// TIA Portal V20 export
FUNCTION_BLOCK "LER_AlignThetaCalibration"   // FB101, LAD
// stored: Access Published, MemoryReserve 100, SetENOAutomatically false
   VAR_INPUT
      enable : Bool;
      cmdComplete : Bool;
      AxisXHomePos { ExternalAccessible := 'False'; ExternalVisible := 'False'; ExternalWritable := 'False'} : LReal;
      AxisY1HomePos { ExternalAccessible := 'False'; ExternalVisible := 'False'; ExternalWritable := 'False'} : LReal;
      AxisY2HomePos { ExternalAccessible := 'False'; ExternalVisible := 'False'; ExternalWritable := 'False'} : LReal;
   END_VAR
   VAR_OUTPUT
      Visiontrigger : Bool;
      cmdRequest : Bool;
      error : Bool;
      busy : Bool;
      done : Bool;
      status : Word;
      CmdNummber : DInt;
      CmdParameter1 : DInt;
      CmdParameter2 : DInt;
      CmdParameter3 : DInt;
   END_VAR
   VAR_IN_OUT
      moduleInterface : "LER_typeAlignThetaCalibrationInterface";
      AlignTableAxisX : DB_ANY;
      AlignTableAxisY1 : DB_ANY;
      AlignTableAxisY2 : DB_ANY;
   END_VAR
   VAR
      statAxisXMovePosition : Array[0..18] of LReal;
      statAxisY1MovePosition : Array[0..18] of LReal;
      statAxisY2MovePosition : Array[0..18] of LReal;
      instAlignTableAxisXMCMoveAbs : MC_MOVEABSOLUTE;
      instAlignTableAxisY1MCMoveAbs { S7_SetPoint := 'True'} : MC_MOVEABSOLUTE;
      instAlignTableAxisY2MCMoveAbs { S7_SetPoint := 'True'} : MC_MOVEABSOLUTE;
      statPulse { S7_SetPoint := 'True'} : Array[1..50] of Bool;
      statMoveXCmd : Array[1..10] of Bool;
      statMoveY1Cmd : Array[1..10] of Bool;
      statMoveY2Cmd : Array[1..10] of Bool;
      statVisionCmd : Array[1..10] of Bool;
      statRequstCmd : Array[1..20] of Bool;
      statTimer : Array[1..50] of TON_TIME;
      statAllMoveSeq : DInt;
      statManualMove : Bool;
      statCmdNummber : DInt;
      statCmdParameter1 : DInt;
      statCmdParameter2 : DInt;
      statCmdParameter3 : DInt;
      statPreSeq : DInt;
      statSeqTimeTonTimer : TON_TIME;
   END_VAR
   VAR_TEMP
      tempAlignTableAxisX : REF_TO TO_SynchronousAxis;
      tempAlignTableAxisY1 : REF_TO TO_SynchronousAxis;
      tempAlignTableAxisY2 : REF_TO TO_SynchronousAxis;
      tempAlignTableAxisXPosition : DInt;
      tempAlignTableAxisY1Position : DInt;
      tempAlignTableAxisY2Position : DInt;
   END_VAR
   VAR CONSTANT
      VISION_DELAY_TIME : Time := T#500ms;
      REQ_DELAY_TIME : Time := T#100ms;
   END_VAR
   VAR_TEMP   // added for the SCL form of the ladder/FBD networks
      _w1 : Bool;
      _w2 : Bool;
      _w3 : Bool;
      _w4 : Bool;
      _w5 : Bool;
      _w6 : Bool;
      _w7 : Bool;
      _w8 : Bool;
      _w9 : Bool;
   END_VAR
BEGIN

REGION Network 1 (SCL): Axis Config
   #tempAlignTableAxisX ?= #AlignTableAxisX;
   #tempAlignTableAxisY1 ?= #AlignTableAxisY1;
   #tempAlignTableAxisY2 ?= #AlignTableAxisY2;
END_REGION

REGION Network 2: Teaching Position Config
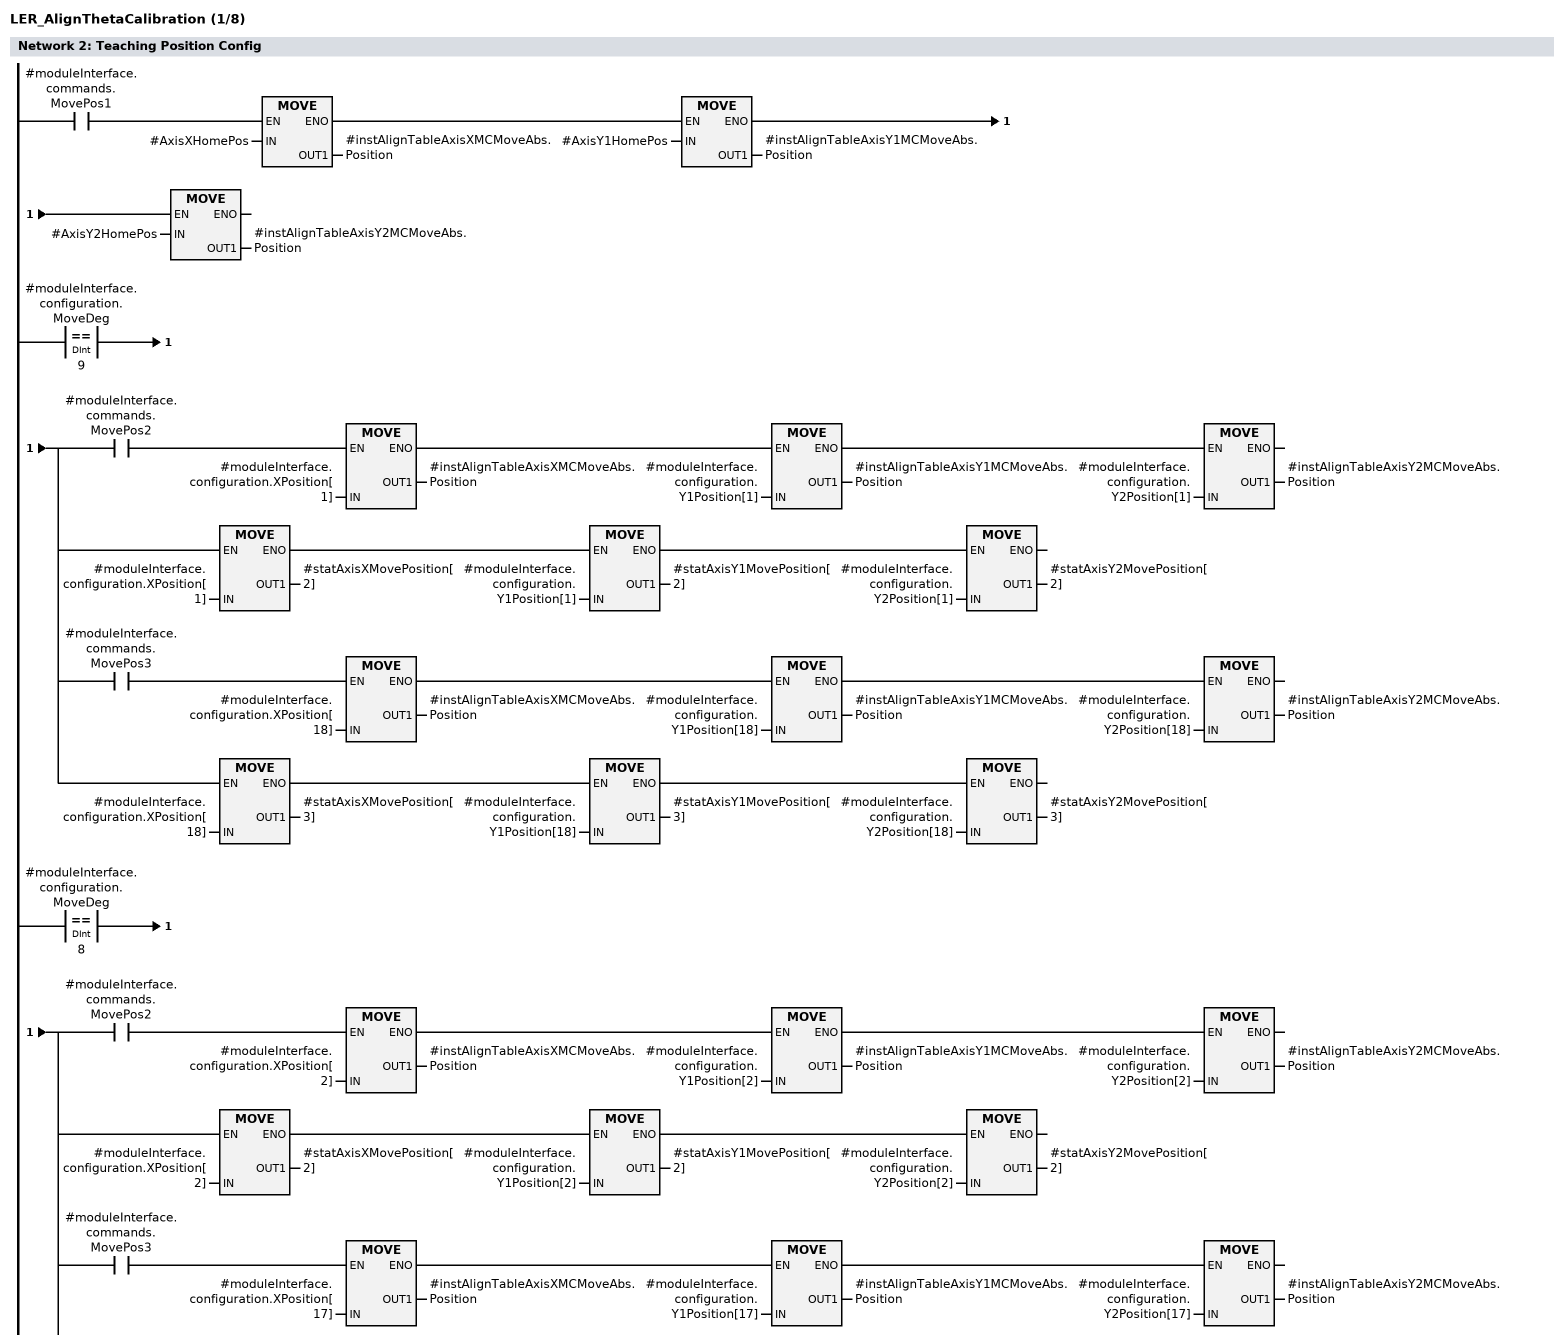
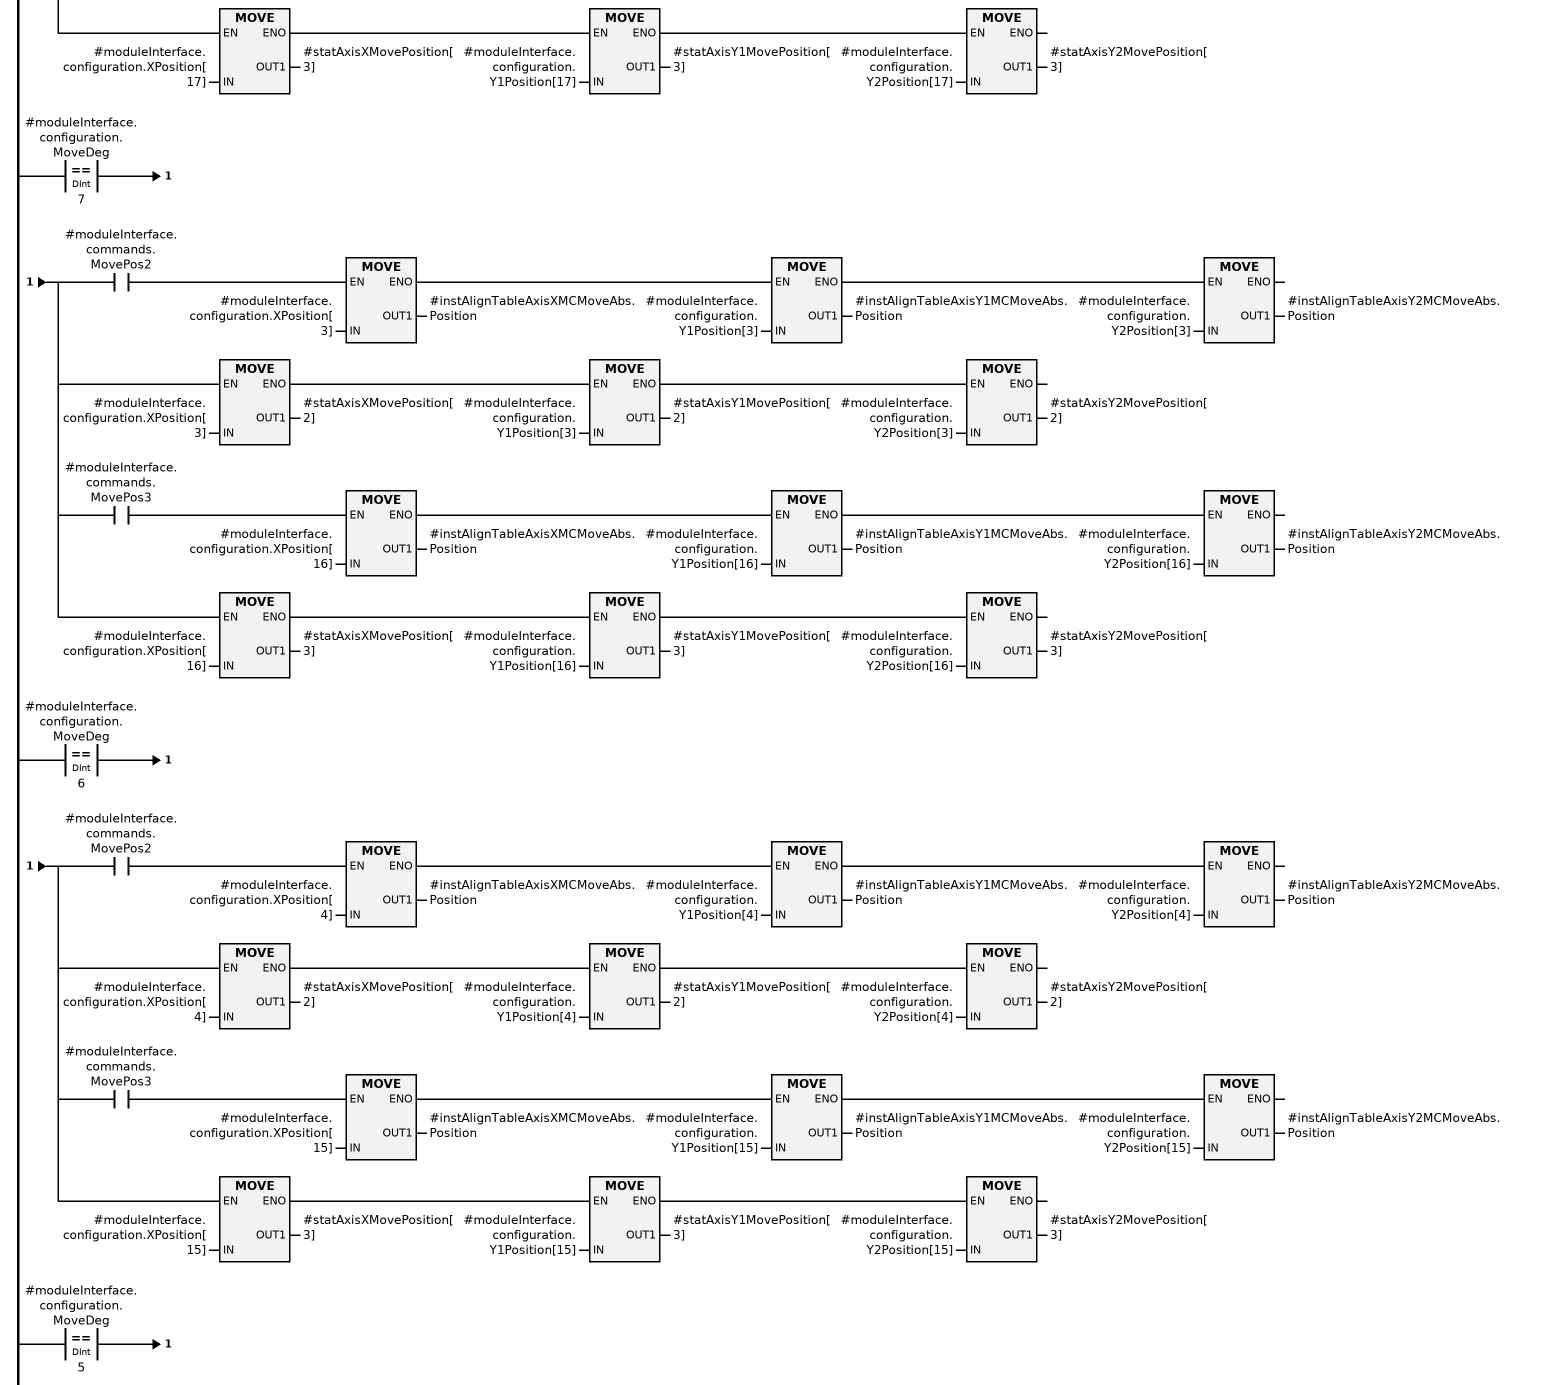
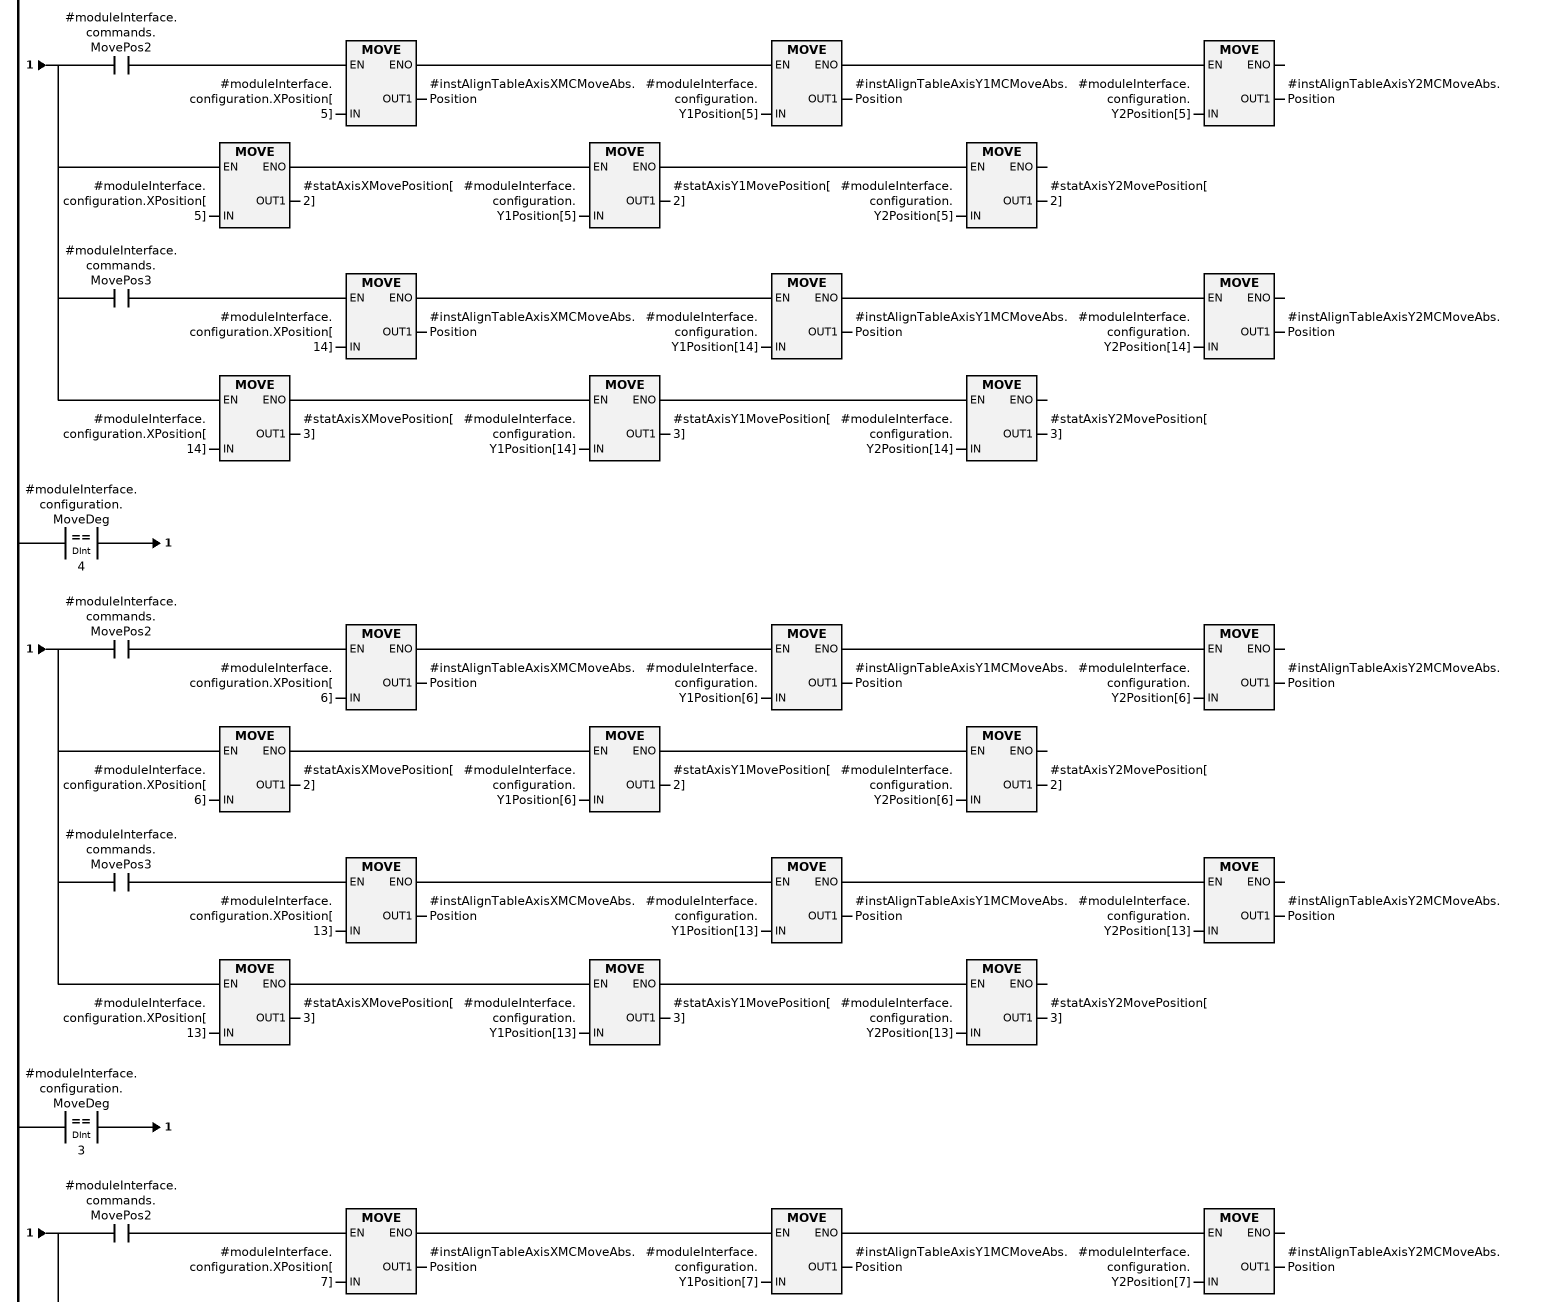
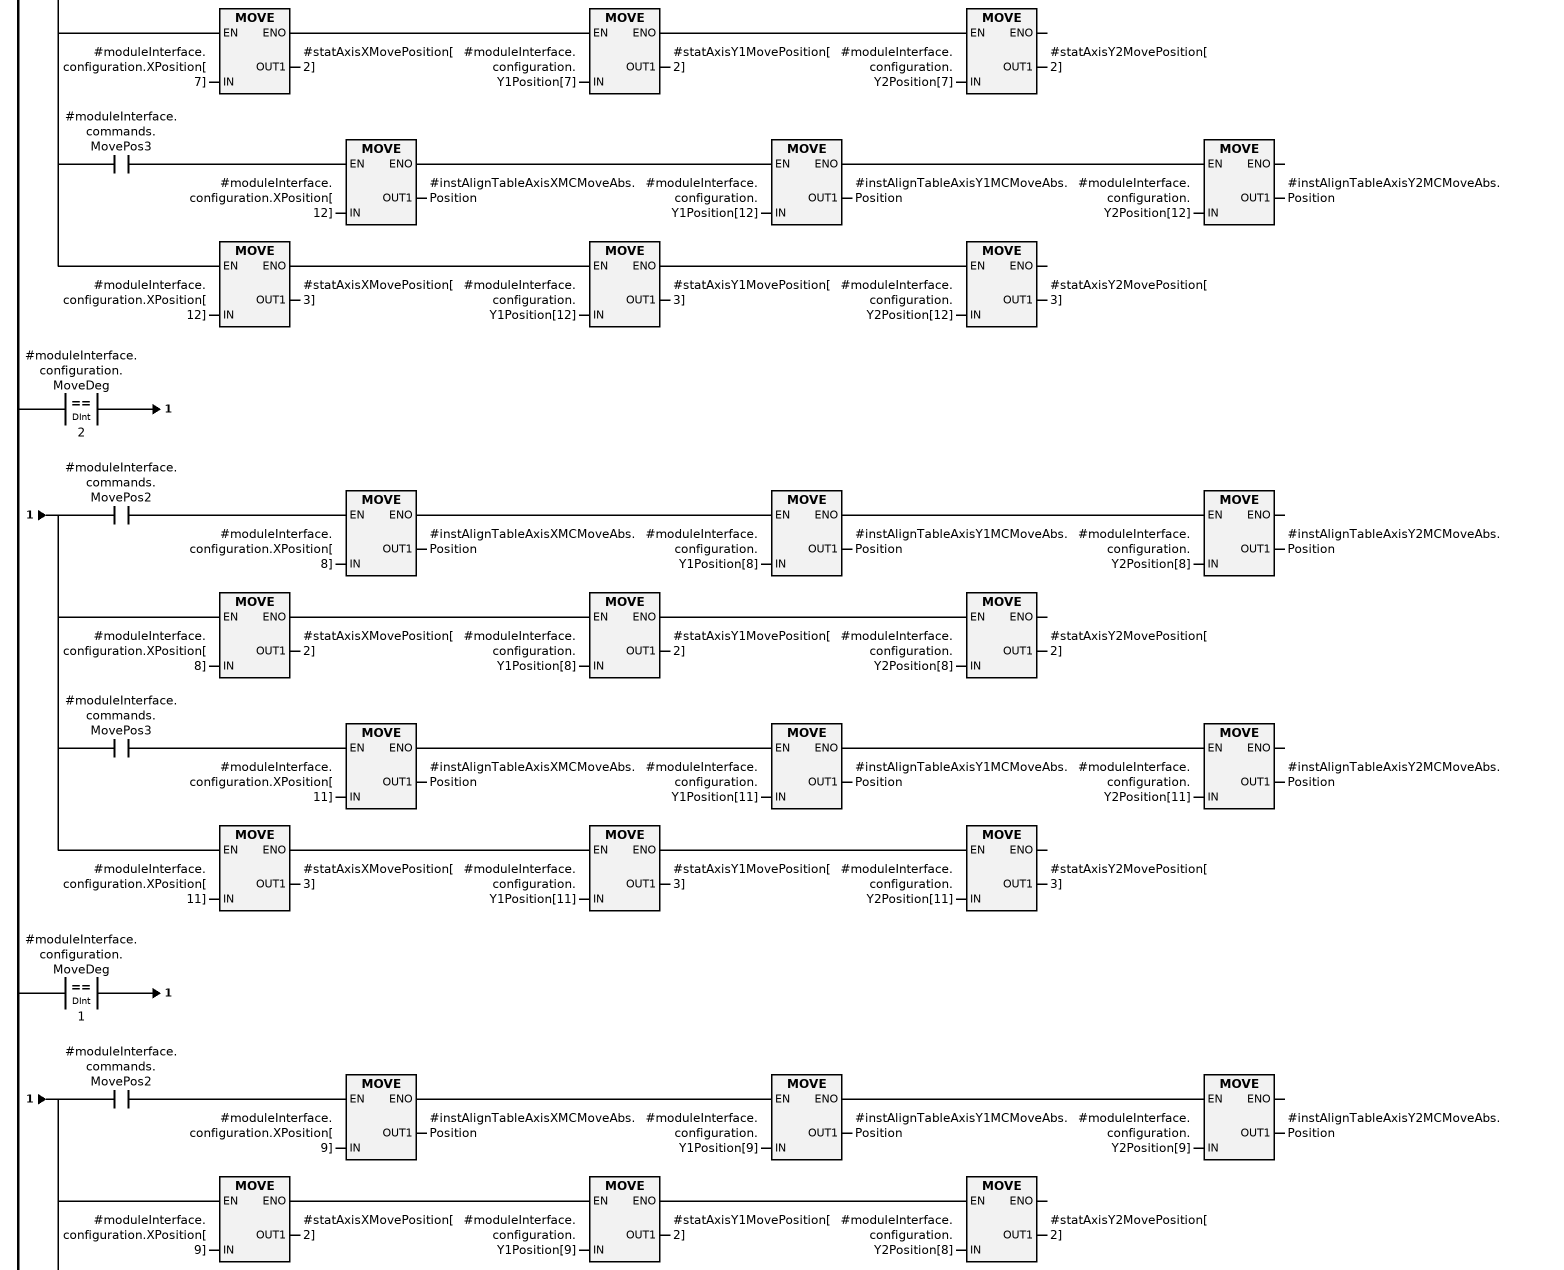
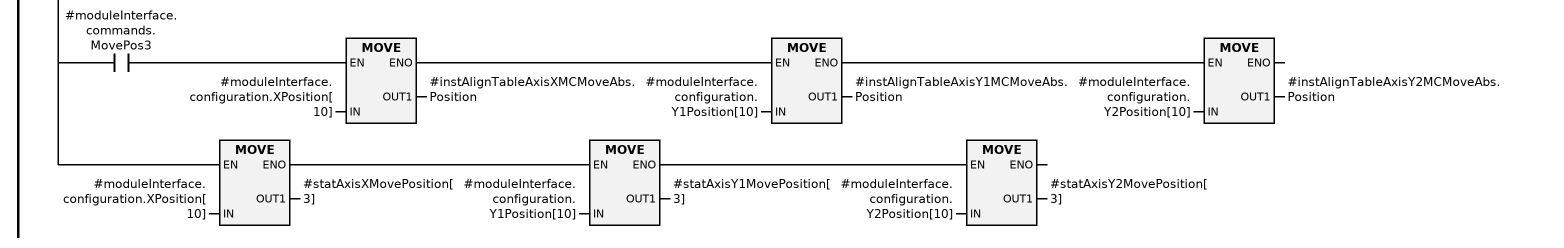
   RUNG wire#powerrail
      Contact( #moduleInterface.commands.MovePos1 )
      Move(in := #AxisXHomePos, out1 => #instAlignTableAxisXMCMoveAbs.Position)
      Move(in := #AxisY1HomePos, out1 => #instAlignTableAxisY1MCMoveAbs.Position)
      Move(in := #AxisY2HomePos, out1 => #instAlignTableAxisY2MCMoveAbs.Position)
   END_RUNG
   RUNG wire#powerrail
      { S7_Templates := "SrcType := DInt" } EQ_Contact(in1 := #moduleInterface.configuration.MoveDeg, in2 := 9)
      wire#w1
      Contact( #moduleInterface.commands.MovePos2 )
      Move(in := #moduleInterface.configuration.XPosition[1], out1 => #instAlignTableAxisXMCMoveAbs.Position)
      Move(in := #moduleInterface.configuration.Y1Position[1], out1 => #instAlignTableAxisY1MCMoveAbs.Position)
      Move(in := #moduleInterface.configuration.Y2Position[1], out1 => #instAlignTableAxisY2MCMoveAbs.Position)
   END_RUNG
   RUNG wire#w1
      Move(in := #moduleInterface.configuration.XPosition[1], out1 => #statAxisXMovePosition[2])
      Move(in := #moduleInterface.configuration.Y1Position[1], out1 => #statAxisY1MovePosition[2])
      Move(in := #moduleInterface.configuration.Y2Position[1], out1 => #statAxisY2MovePosition[2])
   END_RUNG
   RUNG wire#w1
      Contact( #moduleInterface.commands.MovePos3 )
      Move(in := #moduleInterface.configuration.XPosition[18], out1 => #instAlignTableAxisXMCMoveAbs.Position)
      Move(in := #moduleInterface.configuration.Y1Position[18], out1 => #instAlignTableAxisY1MCMoveAbs.Position)
      Move(in := #moduleInterface.configuration.Y2Position[18], out1 => #instAlignTableAxisY2MCMoveAbs.Position)
   END_RUNG
   RUNG wire#w1
      Move(in := #moduleInterface.configuration.XPosition[18], out1 => #statAxisXMovePosition[3])
      Move(in := #moduleInterface.configuration.Y1Position[18], out1 => #statAxisY1MovePosition[3])
      Move(in := #moduleInterface.configuration.Y2Position[18], out1 => #statAxisY2MovePosition[3])
   END_RUNG
   RUNG wire#powerrail
      { S7_Templates := "SrcType := DInt" } EQ_Contact(in1 := #moduleInterface.configuration.MoveDeg, in2 := 8)
      wire#w2
      Contact( #moduleInterface.commands.MovePos2 )
      Move(in := #moduleInterface.configuration.XPosition[2], out1 => #instAlignTableAxisXMCMoveAbs.Position)
      Move(in := #moduleInterface.configuration.Y1Position[2], out1 => #instAlignTableAxisY1MCMoveAbs.Position)
      Move(in := #moduleInterface.configuration.Y2Position[2], out1 => #instAlignTableAxisY2MCMoveAbs.Position)
   END_RUNG
   RUNG wire#w2
      Move(in := #moduleInterface.configuration.XPosition[2], out1 => #statAxisXMovePosition[2])
      Move(in := #moduleInterface.configuration.Y1Position[2], out1 => #statAxisY1MovePosition[2])
      Move(in := #moduleInterface.configuration.Y2Position[2], out1 => #statAxisY2MovePosition[2])
   END_RUNG
   RUNG wire#w2
      Contact( #moduleInterface.commands.MovePos3 )
      Move(in := #moduleInterface.configuration.XPosition[17], out1 => #instAlignTableAxisXMCMoveAbs.Position)
      Move(in := #moduleInterface.configuration.Y1Position[17], out1 => #instAlignTableAxisY1MCMoveAbs.Position)
      Move(in := #moduleInterface.configuration.Y2Position[17], out1 => #instAlignTableAxisY2MCMoveAbs.Position)
   END_RUNG
   RUNG wire#w2
      Move(in := #moduleInterface.configuration.XPosition[17], out1 => #statAxisXMovePosition[3])
      Move(in := #moduleInterface.configuration.Y1Position[17], out1 => #statAxisY1MovePosition[3])
      Move(in := #moduleInterface.configuration.Y2Position[17], out1 => #statAxisY2MovePosition[3])
   END_RUNG
   RUNG wire#powerrail
      { S7_Templates := "SrcType := DInt" } EQ_Contact(in1 := #moduleInterface.configuration.MoveDeg, in2 := 7)
      wire#w3
      Contact( #moduleInterface.commands.MovePos2 )
      Move(in := #moduleInterface.configuration.XPosition[3], out1 => #instAlignTableAxisXMCMoveAbs.Position)
      Move(in := #moduleInterface.configuration.Y1Position[3], out1 => #instAlignTableAxisY1MCMoveAbs.Position)
      Move(in := #moduleInterface.configuration.Y2Position[3], out1 => #instAlignTableAxisY2MCMoveAbs.Position)
   END_RUNG
   RUNG wire#w3
      Move(in := #moduleInterface.configuration.XPosition[3], out1 => #statAxisXMovePosition[2])
      Move(in := #moduleInterface.configuration.Y1Position[3], out1 => #statAxisY1MovePosition[2])
      Move(in := #moduleInterface.configuration.Y2Position[3], out1 => #statAxisY2MovePosition[2])
   END_RUNG
   RUNG wire#w3
      Contact( #moduleInterface.commands.MovePos3 )
      Move(in := #moduleInterface.configuration.XPosition[16], out1 => #instAlignTableAxisXMCMoveAbs.Position)
      Move(in := #moduleInterface.configuration.Y1Position[16], out1 => #instAlignTableAxisY1MCMoveAbs.Position)
      Move(in := #moduleInterface.configuration.Y2Position[16], out1 => #instAlignTableAxisY2MCMoveAbs.Position)
   END_RUNG
   RUNG wire#w3
      Move(in := #moduleInterface.configuration.XPosition[16], out1 => #statAxisXMovePosition[3])
      Move(in := #moduleInterface.configuration.Y1Position[16], out1 => #statAxisY1MovePosition[3])
      Move(in := #moduleInterface.configuration.Y2Position[16], out1 => #statAxisY2MovePosition[3])
   END_RUNG
   RUNG wire#powerrail
      { S7_Templates := "SrcType := DInt" } EQ_Contact(in1 := #moduleInterface.configuration.MoveDeg, in2 := 6)
      wire#w4
      Contact( #moduleInterface.commands.MovePos2 )
      Move(in := #moduleInterface.configuration.XPosition[4], out1 => #instAlignTableAxisXMCMoveAbs.Position)
      Move(in := #moduleInterface.configuration.Y1Position[4], out1 => #instAlignTableAxisY1MCMoveAbs.Position)
      Move(in := #moduleInterface.configuration.Y2Position[4], out1 => #instAlignTableAxisY2MCMoveAbs.Position)
   END_RUNG
   RUNG wire#w4
      Move(in := #moduleInterface.configuration.XPosition[4], out1 => #statAxisXMovePosition[2])
      Move(in := #moduleInterface.configuration.Y1Position[4], out1 => #statAxisY1MovePosition[2])
      Move(in := #moduleInterface.configuration.Y2Position[4], out1 => #statAxisY2MovePosition[2])
   END_RUNG
   RUNG wire#w4
      Contact( #moduleInterface.commands.MovePos3 )
      Move(in := #moduleInterface.configuration.XPosition[15], out1 => #instAlignTableAxisXMCMoveAbs.Position)
      Move(in := #moduleInterface.configuration.Y1Position[15], out1 => #instAlignTableAxisY1MCMoveAbs.Position)
      Move(in := #moduleInterface.configuration.Y2Position[15], out1 => #instAlignTableAxisY2MCMoveAbs.Position)
   END_RUNG
   RUNG wire#w4
      Move(in := #moduleInterface.configuration.XPosition[15], out1 => #statAxisXMovePosition[3])
      Move(in := #moduleInterface.configuration.Y1Position[15], out1 => #statAxisY1MovePosition[3])
      Move(in := #moduleInterface.configuration.Y2Position[15], out1 => #statAxisY2MovePosition[3])
   END_RUNG
   RUNG wire#powerrail
      { S7_Templates := "SrcType := DInt" } EQ_Contact(in1 := #moduleInterface.configuration.MoveDeg, in2 := 5)
      wire#w5
      Contact( #moduleInterface.commands.MovePos2 )
      Move(in := #moduleInterface.configuration.XPosition[5], out1 => #instAlignTableAxisXMCMoveAbs.Position)
      Move(in := #moduleInterface.configuration.Y1Position[5], out1 => #instAlignTableAxisY1MCMoveAbs.Position)
      Move(in := #moduleInterface.configuration.Y2Position[5], out1 => #instAlignTableAxisY2MCMoveAbs.Position)
   END_RUNG
   RUNG wire#w5
      Move(in := #moduleInterface.configuration.XPosition[5], out1 => #statAxisXMovePosition[2])
      Move(in := #moduleInterface.configuration.Y1Position[5], out1 => #statAxisY1MovePosition[2])
      Move(in := #moduleInterface.configuration.Y2Position[5], out1 => #statAxisY2MovePosition[2])
   END_RUNG
   RUNG wire#w5
      Contact( #moduleInterface.commands.MovePos3 )
      Move(in := #moduleInterface.configuration.XPosition[14], out1 => #instAlignTableAxisXMCMoveAbs.Position)
      Move(in := #moduleInterface.configuration.Y1Position[14], out1 => #instAlignTableAxisY1MCMoveAbs.Position)
      Move(in := #moduleInterface.configuration.Y2Position[14], out1 => #instAlignTableAxisY2MCMoveAbs.Position)
   END_RUNG
   RUNG wire#w5
      Move(in := #moduleInterface.configuration.XPosition[14], out1 => #statAxisXMovePosition[3])
      Move(in := #moduleInterface.configuration.Y1Position[14], out1 => #statAxisY1MovePosition[3])
      Move(in := #moduleInterface.configuration.Y2Position[14], out1 => #statAxisY2MovePosition[3])
   END_RUNG
   RUNG wire#powerrail
      { S7_Templates := "SrcType := DInt" } EQ_Contact(in1 := #moduleInterface.configuration.MoveDeg, in2 := 4)
      wire#w6
      Contact( #moduleInterface.commands.MovePos2 )
      Move(in := #moduleInterface.configuration.XPosition[6], out1 => #instAlignTableAxisXMCMoveAbs.Position)
      Move(in := #moduleInterface.configuration.Y1Position[6], out1 => #instAlignTableAxisY1MCMoveAbs.Position)
      Move(in := #moduleInterface.configuration.Y2Position[6], out1 => #instAlignTableAxisY2MCMoveAbs.Position)
   END_RUNG
   RUNG wire#w6
      Move(in := #moduleInterface.configuration.XPosition[6], out1 => #statAxisXMovePosition[2])
      Move(in := #moduleInterface.configuration.Y1Position[6], out1 => #statAxisY1MovePosition[2])
      Move(in := #moduleInterface.configuration.Y2Position[6], out1 => #statAxisY2MovePosition[2])
   END_RUNG
   RUNG wire#w6
      Contact( #moduleInterface.commands.MovePos3 )
      Move(in := #moduleInterface.configuration.XPosition[13], out1 => #instAlignTableAxisXMCMoveAbs.Position)
      Move(in := #moduleInterface.configuration.Y1Position[13], out1 => #instAlignTableAxisY1MCMoveAbs.Position)
      Move(in := #moduleInterface.configuration.Y2Position[13], out1 => #instAlignTableAxisY2MCMoveAbs.Position)
   END_RUNG
   RUNG wire#w6
      Move(in := #moduleInterface.configuration.XPosition[13], out1 => #statAxisXMovePosition[3])
      Move(in := #moduleInterface.configuration.Y1Position[13], out1 => #statAxisY1MovePosition[3])
      Move(in := #moduleInterface.configuration.Y2Position[13], out1 => #statAxisY2MovePosition[3])
   END_RUNG
   RUNG wire#powerrail
      { S7_Templates := "SrcType := DInt" } EQ_Contact(in1 := #moduleInterface.configuration.MoveDeg, in2 := 3)
      wire#w7
      Contact( #moduleInterface.commands.MovePos2 )
      Move(in := #moduleInterface.configuration.XPosition[7], out1 => #instAlignTableAxisXMCMoveAbs.Position)
      Move(in := #moduleInterface.configuration.Y1Position[7], out1 => #instAlignTableAxisY1MCMoveAbs.Position)
      Move(in := #moduleInterface.configuration.Y2Position[7], out1 => #instAlignTableAxisY2MCMoveAbs.Position)
   END_RUNG
   RUNG wire#w7
      Move(in := #moduleInterface.configuration.XPosition[7], out1 => #statAxisXMovePosition[2])
      Move(in := #moduleInterface.configuration.Y1Position[7], out1 => #statAxisY1MovePosition[2])
      Move(in := #moduleInterface.configuration.Y2Position[7], out1 => #statAxisY2MovePosition[2])
   END_RUNG
   RUNG wire#w7
      Contact( #moduleInterface.commands.MovePos3 )
      Move(in := #moduleInterface.configuration.XPosition[12], out1 => #instAlignTableAxisXMCMoveAbs.Position)
      Move(in := #moduleInterface.configuration.Y1Position[12], out1 => #instAlignTableAxisY1MCMoveAbs.Position)
      Move(in := #moduleInterface.configuration.Y2Position[12], out1 => #instAlignTableAxisY2MCMoveAbs.Position)
   END_RUNG
   RUNG wire#w7
      Move(in := #moduleInterface.configuration.XPosition[12], out1 => #statAxisXMovePosition[3])
      Move(in := #moduleInterface.configuration.Y1Position[12], out1 => #statAxisY1MovePosition[3])
      Move(in := #moduleInterface.configuration.Y2Position[12], out1 => #statAxisY2MovePosition[3])
   END_RUNG
   RUNG wire#powerrail
      { S7_Templates := "SrcType := DInt" } EQ_Contact(in1 := #moduleInterface.configuration.MoveDeg, in2 := 2)
      wire#w8
      Contact( #moduleInterface.commands.MovePos2 )
      Move(in := #moduleInterface.configuration.XPosition[8], out1 => #instAlignTableAxisXMCMoveAbs.Position)
      Move(in := #moduleInterface.configuration.Y1Position[8], out1 => #instAlignTableAxisY1MCMoveAbs.Position)
      Move(in := #moduleInterface.configuration.Y2Position[8], out1 => #instAlignTableAxisY2MCMoveAbs.Position)
   END_RUNG
   RUNG wire#w8
      Move(in := #moduleInterface.configuration.XPosition[8], out1 => #statAxisXMovePosition[2])
      Move(in := #moduleInterface.configuration.Y1Position[8], out1 => #statAxisY1MovePosition[2])
      Move(in := #moduleInterface.configuration.Y2Position[8], out1 => #statAxisY2MovePosition[2])
   END_RUNG
   RUNG wire#w8
      Contact( #moduleInterface.commands.MovePos3 )
      Move(in := #moduleInterface.configuration.XPosition[11], out1 => #instAlignTableAxisXMCMoveAbs.Position)
      Move(in := #moduleInterface.configuration.Y1Position[11], out1 => #instAlignTableAxisY1MCMoveAbs.Position)
      Move(in := #moduleInterface.configuration.Y2Position[11], out1 => #instAlignTableAxisY2MCMoveAbs.Position)
   END_RUNG
   RUNG wire#w8
      Move(in := #moduleInterface.configuration.XPosition[11], out1 => #statAxisXMovePosition[3])
      Move(in := #moduleInterface.configuration.Y1Position[11], out1 => #statAxisY1MovePosition[3])
      Move(in := #moduleInterface.configuration.Y2Position[11], out1 => #statAxisY2MovePosition[3])
   END_RUNG
   RUNG wire#powerrail
      { S7_Templates := "SrcType := DInt" } EQ_Contact(in1 := #moduleInterface.configuration.MoveDeg, in2 := 1)
      wire#w9
      Contact( #moduleInterface.commands.MovePos2 )
      Move(in := #moduleInterface.configuration.XPosition[9], out1 => #instAlignTableAxisXMCMoveAbs.Position)
      Move(in := #moduleInterface.configuration.Y1Position[9], out1 => #instAlignTableAxisY1MCMoveAbs.Position)
      Move(in := #moduleInterface.configuration.Y2Position[9], out1 => #instAlignTableAxisY2MCMoveAbs.Position)
   END_RUNG
   RUNG wire#w9
      Move(in := #moduleInterface.configuration.XPosition[9], out1 => #statAxisXMovePosition[2])
      Move(in := #moduleInterface.configuration.Y1Position[9], out1 => #statAxisY1MovePosition[2])
      Move(in := #moduleInterface.configuration.Y2Position[8], out1 => #statAxisY2MovePosition[2])
   END_RUNG
   RUNG wire#w9
      Contact( #moduleInterface.commands.MovePos3 )
      Move(in := #moduleInterface.configuration.XPosition[10], out1 => #instAlignTableAxisXMCMoveAbs.Position)
      Move(in := #moduleInterface.configuration.Y1Position[10], out1 => #instAlignTableAxisY1MCMoveAbs.Position)
      Move(in := #moduleInterface.configuration.Y2Position[10], out1 => #instAlignTableAxisY2MCMoveAbs.Position)
   END_RUNG
   RUNG wire#w9
      Move(in := #moduleInterface.configuration.XPosition[10], out1 => #statAxisXMovePosition[3])
      Move(in := #moduleInterface.configuration.Y1Position[10], out1 => #statAxisY1MovePosition[3])
      Move(in := #moduleInterface.configuration.Y2Position[10], out1 => #statAxisY2MovePosition[3])
   END_RUNG
   // the same network as SCL:
   IF #moduleInterface.commands.MovePos1 THEN
       #instAlignTableAxisXMCMoveAbs.Position := #AxisXHomePos;
       #instAlignTableAxisY1MCMoveAbs.Position := #AxisY1HomePos;
       #instAlignTableAxisY2MCMoveAbs.Position := #AxisY2HomePos;
   END_IF;
   #_w1 := #moduleInterface.configuration.MoveDeg = 9;
   IF #_w1 AND #moduleInterface.commands.MovePos2 THEN
       #instAlignTableAxisXMCMoveAbs.Position := #moduleInterface.configuration.XPosition[1];
       #instAlignTableAxisY1MCMoveAbs.Position := #moduleInterface.configuration.Y1Position[1];
       #instAlignTableAxisY2MCMoveAbs.Position := #moduleInterface.configuration.Y2Position[1];
   END_IF;
   IF #_w1 THEN
       #statAxisXMovePosition[2] := #moduleInterface.configuration.XPosition[1];
       #statAxisY1MovePosition[2] := #moduleInterface.configuration.Y1Position[1];
       #statAxisY2MovePosition[2] := #moduleInterface.configuration.Y2Position[1];
   END_IF;
   IF #_w1 AND #moduleInterface.commands.MovePos3 THEN
       #instAlignTableAxisXMCMoveAbs.Position := #moduleInterface.configuration.XPosition[18];
       #instAlignTableAxisY1MCMoveAbs.Position := #moduleInterface.configuration.Y1Position[18];
       #instAlignTableAxisY2MCMoveAbs.Position := #moduleInterface.configuration.Y2Position[18];
   END_IF;
   IF #_w1 THEN
       #statAxisXMovePosition[3] := #moduleInterface.configuration.XPosition[18];
       #statAxisY1MovePosition[3] := #moduleInterface.configuration.Y1Position[18];
       #statAxisY2MovePosition[3] := #moduleInterface.configuration.Y2Position[18];
   END_IF;
   #_w2 := #moduleInterface.configuration.MoveDeg = 8;
   IF #_w2 AND #moduleInterface.commands.MovePos2 THEN
       #instAlignTableAxisXMCMoveAbs.Position := #moduleInterface.configuration.XPosition[2];
       #instAlignTableAxisY1MCMoveAbs.Position := #moduleInterface.configuration.Y1Position[2];
       #instAlignTableAxisY2MCMoveAbs.Position := #moduleInterface.configuration.Y2Position[2];
   END_IF;
   IF #_w2 THEN
       #statAxisXMovePosition[2] := #moduleInterface.configuration.XPosition[2];
       #statAxisY1MovePosition[2] := #moduleInterface.configuration.Y1Position[2];
       #statAxisY2MovePosition[2] := #moduleInterface.configuration.Y2Position[2];
   END_IF;
   IF #_w2 AND #moduleInterface.commands.MovePos3 THEN
       #instAlignTableAxisXMCMoveAbs.Position := #moduleInterface.configuration.XPosition[17];
       #instAlignTableAxisY1MCMoveAbs.Position := #moduleInterface.configuration.Y1Position[17];
       #instAlignTableAxisY2MCMoveAbs.Position := #moduleInterface.configuration.Y2Position[17];
   END_IF;
   IF #_w2 THEN
       #statAxisXMovePosition[3] := #moduleInterface.configuration.XPosition[17];
       #statAxisY1MovePosition[3] := #moduleInterface.configuration.Y1Position[17];
       #statAxisY2MovePosition[3] := #moduleInterface.configuration.Y2Position[17];
   END_IF;
   #_w3 := #moduleInterface.configuration.MoveDeg = 7;
   IF #_w3 AND #moduleInterface.commands.MovePos2 THEN
       #instAlignTableAxisXMCMoveAbs.Position := #moduleInterface.configuration.XPosition[3];
       #instAlignTableAxisY1MCMoveAbs.Position := #moduleInterface.configuration.Y1Position[3];
       #instAlignTableAxisY2MCMoveAbs.Position := #moduleInterface.configuration.Y2Position[3];
   END_IF;
   IF #_w3 THEN
       #statAxisXMovePosition[2] := #moduleInterface.configuration.XPosition[3];
       #statAxisY1MovePosition[2] := #moduleInterface.configuration.Y1Position[3];
       #statAxisY2MovePosition[2] := #moduleInterface.configuration.Y2Position[3];
   END_IF;
   IF #_w3 AND #moduleInterface.commands.MovePos3 THEN
       #instAlignTableAxisXMCMoveAbs.Position := #moduleInterface.configuration.XPosition[16];
       #instAlignTableAxisY1MCMoveAbs.Position := #moduleInterface.configuration.Y1Position[16];
       #instAlignTableAxisY2MCMoveAbs.Position := #moduleInterface.configuration.Y2Position[16];
   END_IF;
   IF #_w3 THEN
       #statAxisXMovePosition[3] := #moduleInterface.configuration.XPosition[16];
       #statAxisY1MovePosition[3] := #moduleInterface.configuration.Y1Position[16];
       #statAxisY2MovePosition[3] := #moduleInterface.configuration.Y2Position[16];
   END_IF;
   #_w4 := #moduleInterface.configuration.MoveDeg = 6;
   IF #_w4 AND #moduleInterface.commands.MovePos2 THEN
       #instAlignTableAxisXMCMoveAbs.Position := #moduleInterface.configuration.XPosition[4];
       #instAlignTableAxisY1MCMoveAbs.Position := #moduleInterface.configuration.Y1Position[4];
       #instAlignTableAxisY2MCMoveAbs.Position := #moduleInterface.configuration.Y2Position[4];
   END_IF;
   IF #_w4 THEN
       #statAxisXMovePosition[2] := #moduleInterface.configuration.XPosition[4];
       #statAxisY1MovePosition[2] := #moduleInterface.configuration.Y1Position[4];
       #statAxisY2MovePosition[2] := #moduleInterface.configuration.Y2Position[4];
   END_IF;
   IF #_w4 AND #moduleInterface.commands.MovePos3 THEN
       #instAlignTableAxisXMCMoveAbs.Position := #moduleInterface.configuration.XPosition[15];
       #instAlignTableAxisY1MCMoveAbs.Position := #moduleInterface.configuration.Y1Position[15];
       #instAlignTableAxisY2MCMoveAbs.Position := #moduleInterface.configuration.Y2Position[15];
   END_IF;
   IF #_w4 THEN
       #statAxisXMovePosition[3] := #moduleInterface.configuration.XPosition[15];
       #statAxisY1MovePosition[3] := #moduleInterface.configuration.Y1Position[15];
       #statAxisY2MovePosition[3] := #moduleInterface.configuration.Y2Position[15];
   END_IF;
   #_w5 := #moduleInterface.configuration.MoveDeg = 5;
   IF #_w5 AND #moduleInterface.commands.MovePos2 THEN
       #instAlignTableAxisXMCMoveAbs.Position := #moduleInterface.configuration.XPosition[5];
       #instAlignTableAxisY1MCMoveAbs.Position := #moduleInterface.configuration.Y1Position[5];
       #instAlignTableAxisY2MCMoveAbs.Position := #moduleInterface.configuration.Y2Position[5];
   END_IF;
   IF #_w5 THEN
       #statAxisXMovePosition[2] := #moduleInterface.configuration.XPosition[5];
       #statAxisY1MovePosition[2] := #moduleInterface.configuration.Y1Position[5];
       #statAxisY2MovePosition[2] := #moduleInterface.configuration.Y2Position[5];
   END_IF;
   IF #_w5 AND #moduleInterface.commands.MovePos3 THEN
       #instAlignTableAxisXMCMoveAbs.Position := #moduleInterface.configuration.XPosition[14];
       #instAlignTableAxisY1MCMoveAbs.Position := #moduleInterface.configuration.Y1Position[14];
       #instAlignTableAxisY2MCMoveAbs.Position := #moduleInterface.configuration.Y2Position[14];
   END_IF;
   IF #_w5 THEN
       #statAxisXMovePosition[3] := #moduleInterface.configuration.XPosition[14];
       #statAxisY1MovePosition[3] := #moduleInterface.configuration.Y1Position[14];
       #statAxisY2MovePosition[3] := #moduleInterface.configuration.Y2Position[14];
   END_IF;
   #_w6 := #moduleInterface.configuration.MoveDeg = 4;
   IF #_w6 AND #moduleInterface.commands.MovePos2 THEN
       #instAlignTableAxisXMCMoveAbs.Position := #moduleInterface.configuration.XPosition[6];
       #instAlignTableAxisY1MCMoveAbs.Position := #moduleInterface.configuration.Y1Position[6];
       #instAlignTableAxisY2MCMoveAbs.Position := #moduleInterface.configuration.Y2Position[6];
   END_IF;
   IF #_w6 THEN
       #statAxisXMovePosition[2] := #moduleInterface.configuration.XPosition[6];
       #statAxisY1MovePosition[2] := #moduleInterface.configuration.Y1Position[6];
       #statAxisY2MovePosition[2] := #moduleInterface.configuration.Y2Position[6];
   END_IF;
   IF #_w6 AND #moduleInterface.commands.MovePos3 THEN
       #instAlignTableAxisXMCMoveAbs.Position := #moduleInterface.configuration.XPosition[13];
       #instAlignTableAxisY1MCMoveAbs.Position := #moduleInterface.configuration.Y1Position[13];
       #instAlignTableAxisY2MCMoveAbs.Position := #moduleInterface.configuration.Y2Position[13];
   END_IF;
   IF #_w6 THEN
       #statAxisXMovePosition[3] := #moduleInterface.configuration.XPosition[13];
       #statAxisY1MovePosition[3] := #moduleInterface.configuration.Y1Position[13];
       #statAxisY2MovePosition[3] := #moduleInterface.configuration.Y2Position[13];
   END_IF;
   #_w7 := #moduleInterface.configuration.MoveDeg = 3;
   IF #_w7 AND #moduleInterface.commands.MovePos2 THEN
       #instAlignTableAxisXMCMoveAbs.Position := #moduleInterface.configuration.XPosition[7];
       #instAlignTableAxisY1MCMoveAbs.Position := #moduleInterface.configuration.Y1Position[7];
       #instAlignTableAxisY2MCMoveAbs.Position := #moduleInterface.configuration.Y2Position[7];
   END_IF;
   IF #_w7 THEN
       #statAxisXMovePosition[2] := #moduleInterface.configuration.XPosition[7];
       #statAxisY1MovePosition[2] := #moduleInterface.configuration.Y1Position[7];
       #statAxisY2MovePosition[2] := #moduleInterface.configuration.Y2Position[7];
   END_IF;
   IF #_w7 AND #moduleInterface.commands.MovePos3 THEN
       #instAlignTableAxisXMCMoveAbs.Position := #moduleInterface.configuration.XPosition[12];
       #instAlignTableAxisY1MCMoveAbs.Position := #moduleInterface.configuration.Y1Position[12];
       #instAlignTableAxisY2MCMoveAbs.Position := #moduleInterface.configuration.Y2Position[12];
   END_IF;
   IF #_w7 THEN
       #statAxisXMovePosition[3] := #moduleInterface.configuration.XPosition[12];
       #statAxisY1MovePosition[3] := #moduleInterface.configuration.Y1Position[12];
       #statAxisY2MovePosition[3] := #moduleInterface.configuration.Y2Position[12];
   END_IF;
   #_w8 := #moduleInterface.configuration.MoveDeg = 2;
   IF #_w8 AND #moduleInterface.commands.MovePos2 THEN
       #instAlignTableAxisXMCMoveAbs.Position := #moduleInterface.configuration.XPosition[8];
       #instAlignTableAxisY1MCMoveAbs.Position := #moduleInterface.configuration.Y1Position[8];
       #instAlignTableAxisY2MCMoveAbs.Position := #moduleInterface.configuration.Y2Position[8];
   END_IF;
   IF #_w8 THEN
       #statAxisXMovePosition[2] := #moduleInterface.configuration.XPosition[8];
       #statAxisY1MovePosition[2] := #moduleInterface.configuration.Y1Position[8];
       #statAxisY2MovePosition[2] := #moduleInterface.configuration.Y2Position[8];
   END_IF;
   IF #_w8 AND #moduleInterface.commands.MovePos3 THEN
       #instAlignTableAxisXMCMoveAbs.Position := #moduleInterface.configuration.XPosition[11];
       #instAlignTableAxisY1MCMoveAbs.Position := #moduleInterface.configuration.Y1Position[11];
       #instAlignTableAxisY2MCMoveAbs.Position := #moduleInterface.configuration.Y2Position[11];
   END_IF;
   IF #_w8 THEN
       #statAxisXMovePosition[3] := #moduleInterface.configuration.XPosition[11];
       #statAxisY1MovePosition[3] := #moduleInterface.configuration.Y1Position[11];
       #statAxisY2MovePosition[3] := #moduleInterface.configuration.Y2Position[11];
   END_IF;
   #_w9 := #moduleInterface.configuration.MoveDeg = 1;
   IF #_w9 AND #moduleInterface.commands.MovePos2 THEN
       #instAlignTableAxisXMCMoveAbs.Position := #moduleInterface.configuration.XPosition[9];
       #instAlignTableAxisY1MCMoveAbs.Position := #moduleInterface.configuration.Y1Position[9];
       #instAlignTableAxisY2MCMoveAbs.Position := #moduleInterface.configuration.Y2Position[9];
   END_IF;
   IF #_w9 THEN
       #statAxisXMovePosition[2] := #moduleInterface.configuration.XPosition[9];
       #statAxisY1MovePosition[2] := #moduleInterface.configuration.Y1Position[9];
       #statAxisY2MovePosition[2] := #moduleInterface.configuration.Y2Position[8];
   END_IF;
   IF #_w9 AND #moduleInterface.commands.MovePos3 THEN
       #instAlignTableAxisXMCMoveAbs.Position := #moduleInterface.configuration.XPosition[10];
       #instAlignTableAxisY1MCMoveAbs.Position := #moduleInterface.configuration.Y1Position[10];
       #instAlignTableAxisY2MCMoveAbs.Position := #moduleInterface.configuration.Y2Position[10];
   END_IF;
   IF #_w9 THEN
       #statAxisXMovePosition[3] := #moduleInterface.configuration.XPosition[10];
       #statAxisY1MovePosition[3] := #moduleInterface.configuration.Y1Position[10];
       #statAxisY2MovePosition[3] := #moduleInterface.configuration.Y2Position[10];
   END_IF;
END_REGION

REGION Network 3: Axis Poistion Config
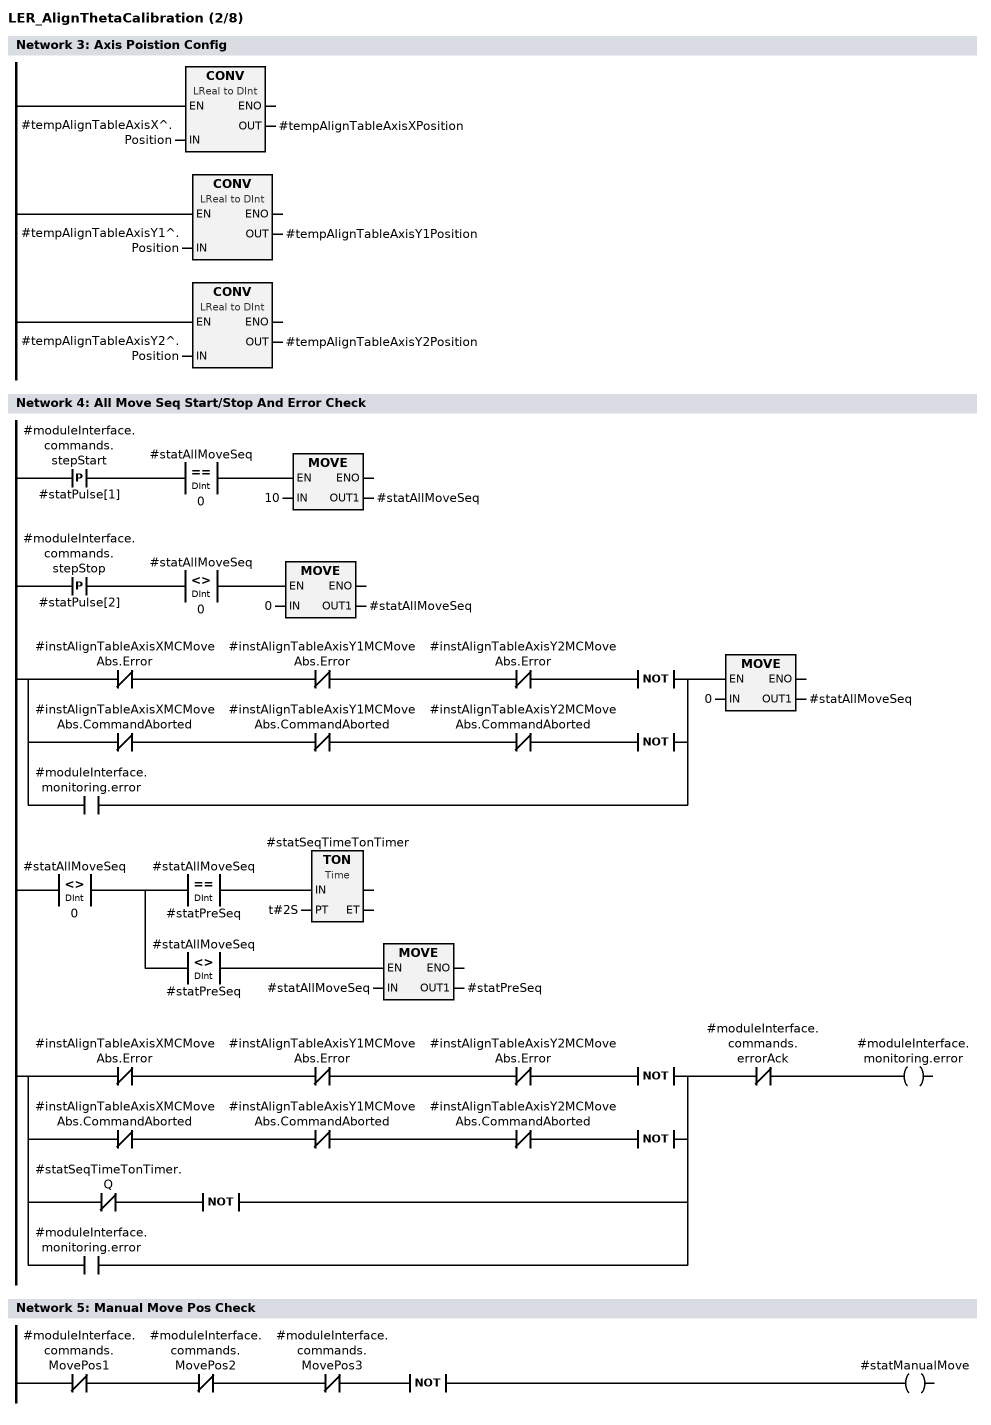
   RUNG wire#powerrail
      { S7_Templates := "[SrcType := LReal, DestType := DInt]" } Convert(in := #tempAlignTableAxisX^.Position, out => #tempAlignTableAxisXPosition)
   END_RUNG
   RUNG wire#powerrail
      { S7_Templates := "[SrcType := LReal, DestType := DInt]" } Convert(in := #tempAlignTableAxisY1^.Position, out => #tempAlignTableAxisY1Position)
   END_RUNG
   RUNG wire#powerrail
      { S7_Templates := "[SrcType := LReal, DestType := DInt]" } Convert(in := #tempAlignTableAxisY2^.Position, out => #tempAlignTableAxisY2Position)
   END_RUNG
   // the same network as SCL:
   #tempAlignTableAxisXPosition := LREAL_TO_DINT(#tempAlignTableAxisX^.Position);
   #tempAlignTableAxisY1Position := LREAL_TO_DINT(#tempAlignTableAxisY1^.Position);
   #tempAlignTableAxisY2Position := LREAL_TO_DINT(#tempAlignTableAxisY2^.Position);
END_REGION

REGION Network 4: All Move Seq Start/Stop And Error Check
   RUNG wire#powerrail
      P_Contact(operand := #moduleInterface.commands.stepStart, bit := #statPulse[1])
      { S7_Templates := "SrcType := DInt" } EQ_Contact(in1 := #statAllMoveSeq, in2 := 0)
      Move(in := 10, out1 => #statAllMoveSeq)
   END_RUNG
   RUNG wire#powerrail
      P_Contact(operand := #moduleInterface.commands.stepStop, bit := #statPulse[2])
      { S7_Templates := "SrcType := DInt" } NE_Contact(in1 := #statAllMoveSeq, in2 := 0)
      Move(in := 0, out1 => #statAllMoveSeq)
   END_RUNG
   RUNG wire#powerrail
      I_Contact( #instAlignTableAxisXMCMoveAbs.Error )
      I_Contact( #instAlignTableAxisY1MCMoveAbs.Error )
      I_Contact( #instAlignTableAxisY2MCMoveAbs.Error )
      Not()
      wire#w1
      Move(in := 0, out1 => #statAllMoveSeq)
   END_RUNG
   RUNG wire#powerrail
      I_Contact( #instAlignTableAxisXMCMoveAbs.CommandAborted )
      I_Contact( #instAlignTableAxisY1MCMoveAbs.CommandAborted )
      I_Contact( #instAlignTableAxisY2MCMoveAbs.CommandAborted )
      Not()
   END_RUNG wire#w1
   RUNG wire#powerrail
      Contact( #moduleInterface.monitoring.error )
   END_RUNG wire#w1
   RUNG wire#powerrail
      { S7_Templates := "SrcType := DInt" } NE_Contact(in1 := #statAllMoveSeq, in2 := 0)
      wire#w2
      { S7_Templates := "SrcType := DInt" } EQ_Contact(in1 := #statAllMoveSeq, in2 := #statPreSeq)
      { S7_Templates := "time_type := Time" } #statSeqTimeTonTimer.TON(pt := t#2S, et =>)
   END_RUNG
   RUNG wire#w2
      { S7_Templates := "SrcType := DInt" } NE_Contact(in1 := #statAllMoveSeq, in2 := #statPreSeq)
      Move(in := #statAllMoveSeq, out1 => #statPreSeq)
   END_RUNG
   RUNG wire#powerrail
      I_Contact( #instAlignTableAxisXMCMoveAbs.Error )
      I_Contact( #instAlignTableAxisY1MCMoveAbs.Error )
      I_Contact( #instAlignTableAxisY2MCMoveAbs.Error )
      Not()
      wire#w3
      I_Contact( #moduleInterface.commands.errorAck )
      Coil( #moduleInterface.monitoring.error )
   END_RUNG
   RUNG wire#powerrail
      I_Contact( #instAlignTableAxisXMCMoveAbs.CommandAborted )
      I_Contact( #instAlignTableAxisY1MCMoveAbs.CommandAborted )
      I_Contact( #instAlignTableAxisY2MCMoveAbs.CommandAborted )
      Not()
   END_RUNG wire#w3
   RUNG wire#powerrail
      I_Contact( #statSeqTimeTonTimer.Q )
      Not()
   END_RUNG wire#w3
   RUNG wire#powerrail
      Contact( #moduleInterface.monitoring.error )
   END_RUNG wire#w3
   // the same network as SCL:
   #_w1 := #moduleInterface.commands.stepStart AND NOT #statPulse[1];   // rising edge of #moduleInterface.commands.stepStart
   #statPulse[1] := #moduleInterface.commands.stepStart;
   IF #_w1 AND (#statAllMoveSeq = 0) THEN #statAllMoveSeq := 10; END_IF;
   #_w2 := #moduleInterface.commands.stepStop AND NOT #statPulse[2];   // rising edge of #moduleInterface.commands.stepStop
   #statPulse[2] := #moduleInterface.commands.stepStop;
   IF #_w2 AND (#statAllMoveSeq <> 0) THEN #statAllMoveSeq := 0; END_IF;
   IF NOT (NOT #instAlignTableAxisXMCMoveAbs.Error AND NOT #instAlignTableAxisY1MCMoveAbs.Error AND NOT #instAlignTableAxisY2MCMoveAbs.Error) OR NOT (NOT #instAlignTableAxisXMCMoveAbs.CommandAborted AND NOT #instAlignTableAxisY1MCMoveAbs.CommandAborted AND NOT #instAlignTableAxisY2MCMoveAbs.CommandAborted) OR #moduleInterface.monitoring.error THEN
       #statAllMoveSeq := 0;
   END_IF;
   #_w3 := #statAllMoveSeq <> 0;
   #statSeqTimeTonTimer(IN := #_w3 AND (#statAllMoveSeq = #statPreSeq), PT := t#2S);   // TON
   IF #_w3 AND (#statAllMoveSeq <> #statPreSeq) THEN #statPreSeq := #statAllMoveSeq; END_IF;
   #moduleInterface.monitoring.error := (NOT (NOT #instAlignTableAxisXMCMoveAbs.Error AND NOT #instAlignTableAxisY1MCMoveAbs.Error AND NOT #instAlignTableAxisY2MCMoveAbs.Error) OR NOT (NOT #instAlignTableAxisXMCMoveAbs.CommandAborted AND NOT #instAlignTableAxisY1MCMoveAbs.CommandAborted AND NOT #instAlignTableAxisY2MCMoveAbs.CommandAborted) OR NOT (NOT #statSeqTimeTonTimer.Q) OR #moduleInterface.monitoring.error) AND NOT #moduleInterface.commands.errorAck;
END_REGION

REGION Network 5: Manual Move Pos Check
   RUNG wire#powerrail
      I_Contact( #moduleInterface.commands.MovePos1 )
      I_Contact( #moduleInterface.commands.MovePos2 )
      I_Contact( #moduleInterface.commands.MovePos3 )
      Not()
      Coil( #statManualMove )
   END_RUNG
   // the same network as SCL:
   #statManualMove := NOT (NOT #moduleInterface.commands.MovePos1 AND NOT #moduleInterface.commands.MovePos2 AND NOT #moduleInterface.commands.MovePos3);
END_REGION

REGION Network 6: === Sequence Start ===
END_REGION

REGION Network 7: All Move Seq Pos 1 [Seq 10]
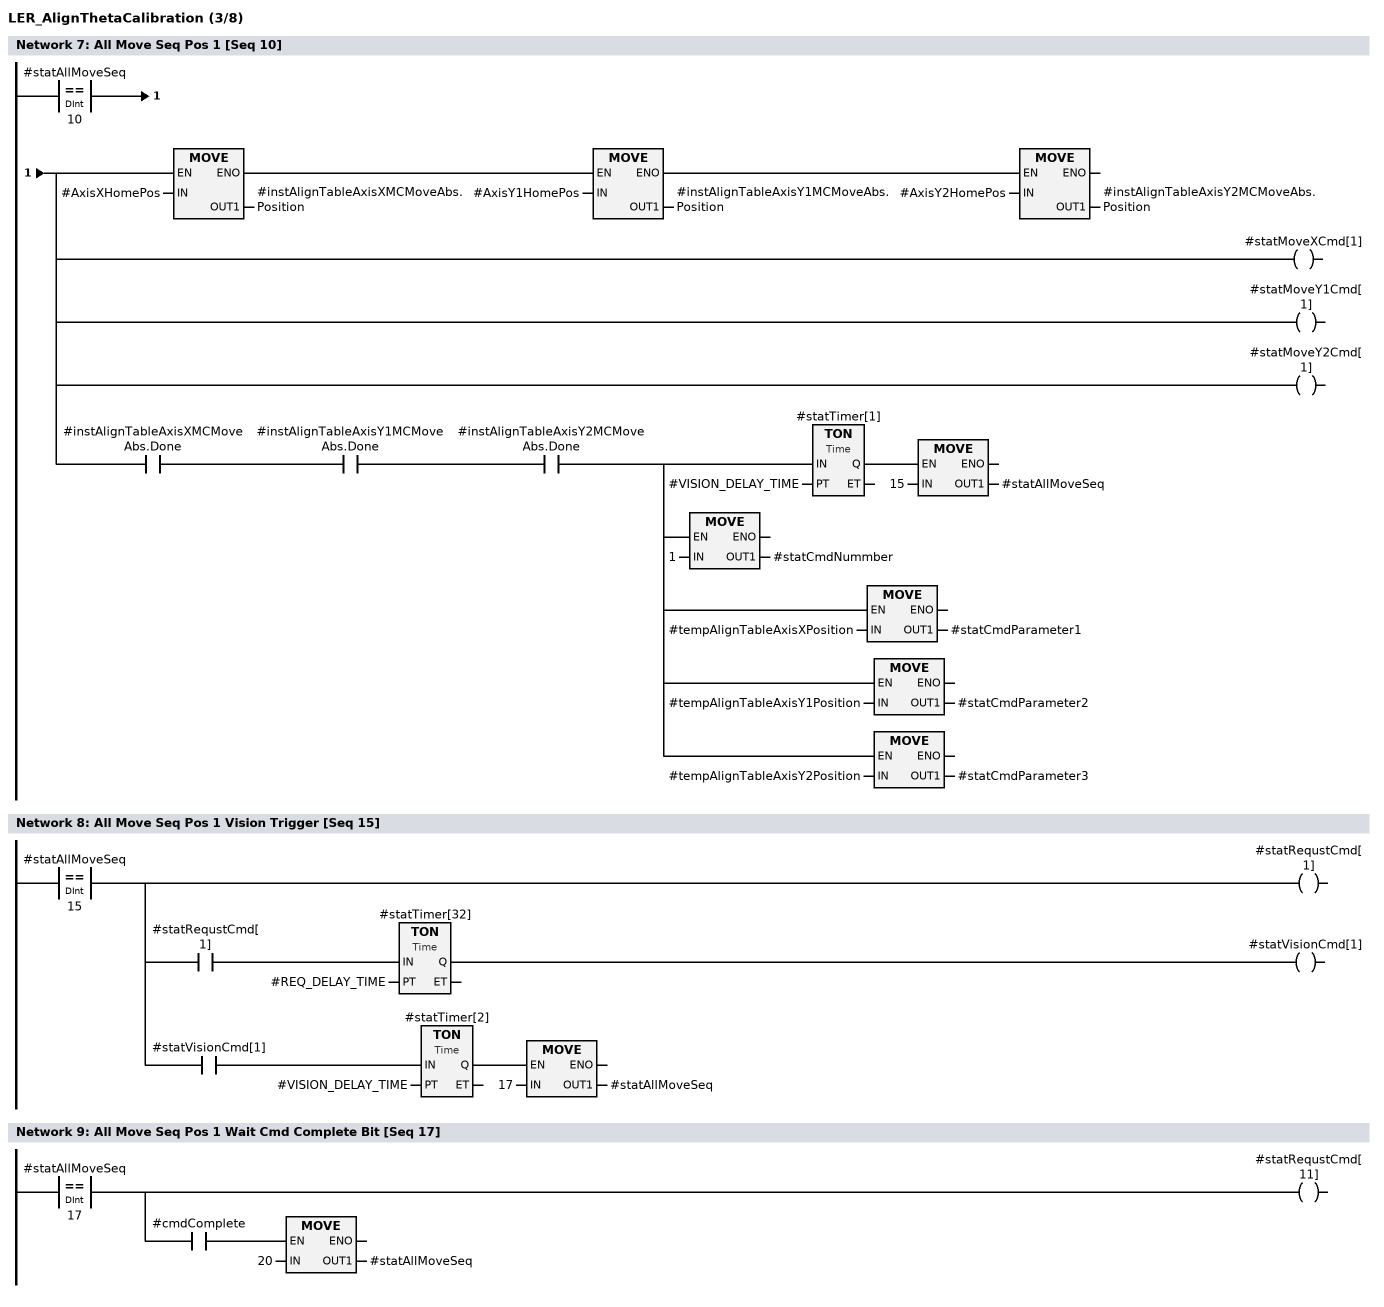
   RUNG wire#powerrail
      { S7_Templates := "SrcType := DInt" } EQ_Contact(in1 := #statAllMoveSeq, in2 := 10)
      wire#w1
      Move(in := #AxisXHomePos, out1 => #instAlignTableAxisXMCMoveAbs.Position)
      Move(in := #AxisY1HomePos, out1 => #instAlignTableAxisY1MCMoveAbs.Position)
      Move(in := #AxisY2HomePos, out1 => #instAlignTableAxisY2MCMoveAbs.Position)
   END_RUNG
   RUNG wire#w1
      Coil( #statMoveXCmd[1] )
   END_RUNG
   RUNG wire#w1
      Coil( #statMoveY1Cmd[1] )
   END_RUNG
   RUNG wire#w1
      Coil( #statMoveY2Cmd[1] )
   END_RUNG
   RUNG wire#w1
      Contact( #instAlignTableAxisXMCMoveAbs.Done )
      Contact( #instAlignTableAxisY1MCMoveAbs.Done )
      Contact( #instAlignTableAxisY2MCMoveAbs.Done )
      wire#w2
      { S7_Templates := "time_type := Time" } #statTimer[1].TON(pt := #VISION_DELAY_TIME, et =>)
      Move(in := 15, out1 => #statAllMoveSeq)
   END_RUNG
   RUNG wire#w2
      Move(in := 1, out1 => #statCmdNummber)
   END_RUNG
   RUNG wire#w2
      Move(in := #tempAlignTableAxisXPosition, out1 => #statCmdParameter1)
   END_RUNG
   RUNG wire#w2
      Move(in := #tempAlignTableAxisY1Position, out1 => #statCmdParameter2)
   END_RUNG
   RUNG wire#w2
      Move(in := #tempAlignTableAxisY2Position, out1 => #statCmdParameter3)
   END_RUNG
   // the same network as SCL:
   #_w1 := #statAllMoveSeq = 10;
   IF #_w1 THEN
       #instAlignTableAxisXMCMoveAbs.Position := #AxisXHomePos;
       #instAlignTableAxisY1MCMoveAbs.Position := #AxisY1HomePos;
       #instAlignTableAxisY2MCMoveAbs.Position := #AxisY2HomePos;
   END_IF;
   #statMoveXCmd[1] := #_w1;
   #statMoveY1Cmd[1] := #_w1;
   #statMoveY2Cmd[1] := #_w1;
   #_w2 := #_w1 AND #instAlignTableAxisXMCMoveAbs.Done AND #instAlignTableAxisY1MCMoveAbs.Done AND #instAlignTableAxisY2MCMoveAbs.Done;
   #statTimer[1].TON(IN := #_w2, PT := #VISION_DELAY_TIME);
   IF #statTimer[1].Q THEN #statAllMoveSeq := 15; END_IF;
   IF #_w2 THEN
       #statCmdNummber := 1;
       #statCmdParameter1 := #tempAlignTableAxisXPosition;
       #statCmdParameter2 := #tempAlignTableAxisY1Position;
       #statCmdParameter3 := #tempAlignTableAxisY2Position;
   END_IF;
END_REGION

REGION Network 8: All Move Seq Pos 1 Vision Trigger [Seq 15]
   RUNG wire#powerrail
      { S7_Templates := "SrcType := DInt" } EQ_Contact(in1 := #statAllMoveSeq, in2 := 15)
      wire#w1
      Coil( #statRequstCmd[1] )
   END_RUNG
   RUNG wire#w1
      Contact( #statRequstCmd[1] )
      { S7_Templates := "time_type := Time" } #statTimer[32].TON(pt := #REQ_DELAY_TIME, et =>)
      Coil( #statVisionCmd[1] )
   END_RUNG
   RUNG wire#w1
      Contact( #statVisionCmd[1] )
      { S7_Templates := "time_type := Time" } #statTimer[2].TON(pt := #VISION_DELAY_TIME, et =>)
      Move(in := 17, out1 => #statAllMoveSeq)
   END_RUNG
   // the same network as SCL:
   #statRequstCmd[1] := #statAllMoveSeq = 15;
   #statTimer[32].TON(IN := (#statAllMoveSeq = 15) AND #statRequstCmd[1], PT := #REQ_DELAY_TIME);
   #statVisionCmd[1] := #statTimer[32].Q;
   #statTimer[2].TON(IN := (#statAllMoveSeq = 15) AND #statVisionCmd[1], PT := #VISION_DELAY_TIME);
   IF #statTimer[2].Q THEN #statAllMoveSeq := 17; END_IF;
END_REGION

REGION Network 9: All Move Seq Pos 1 Wait Cmd Complete Bit [Seq 17]
   RUNG wire#powerrail
      { S7_Templates := "SrcType := DInt" } EQ_Contact(in1 := #statAllMoveSeq, in2 := 17)
      wire#w1
      Coil( #statRequstCmd[11] )
   END_RUNG
   RUNG wire#w1
      Contact( #cmdComplete )
      Move(in := 20, out1 => #statAllMoveSeq)
   END_RUNG
   // the same network as SCL:
   #statRequstCmd[11] := #statAllMoveSeq = 17;
   IF (#statAllMoveSeq = 17) AND #cmdComplete THEN #statAllMoveSeq := 20; END_IF;
END_REGION

REGION Network 10: All Move Seq Pos 2 [Seq 20]
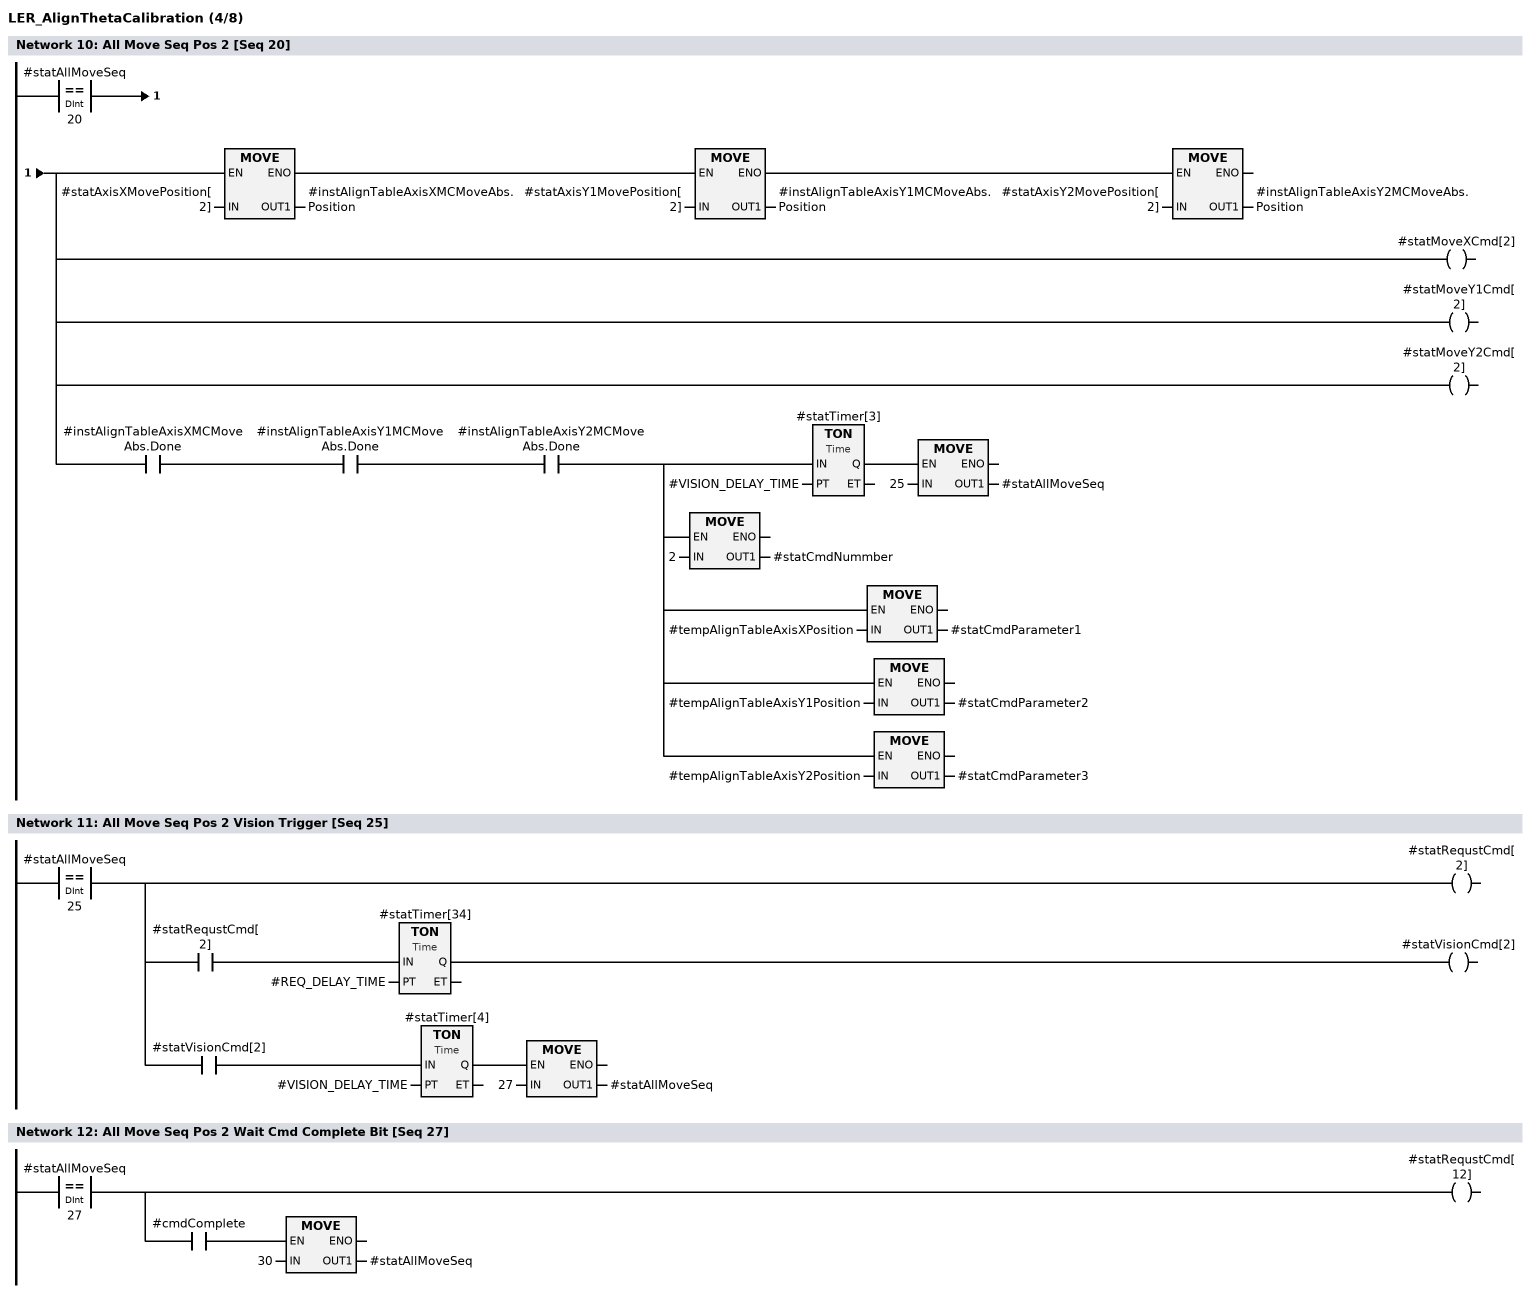
   RUNG wire#powerrail
      { S7_Templates := "SrcType := DInt" } EQ_Contact(in1 := #statAllMoveSeq, in2 := 20)
      wire#w1
      Move(in := #statAxisXMovePosition[2], out1 => #instAlignTableAxisXMCMoveAbs.Position)
      Move(in := #statAxisY1MovePosition[2], out1 => #instAlignTableAxisY1MCMoveAbs.Position)
      Move(in := #statAxisY2MovePosition[2], out1 => #instAlignTableAxisY2MCMoveAbs.Position)
   END_RUNG
   RUNG wire#w1
      Coil( #statMoveXCmd[2] )
   END_RUNG
   RUNG wire#w1
      Coil( #statMoveY1Cmd[2] )
   END_RUNG
   RUNG wire#w1
      Coil( #statMoveY2Cmd[2] )
   END_RUNG
   RUNG wire#w1
      Contact( #instAlignTableAxisXMCMoveAbs.Done )
      Contact( #instAlignTableAxisY1MCMoveAbs.Done )
      Contact( #instAlignTableAxisY2MCMoveAbs.Done )
      wire#w2
      { S7_Templates := "time_type := Time" } #statTimer[3].TON(pt := #VISION_DELAY_TIME, et =>)
      Move(in := 25, out1 => #statAllMoveSeq)
   END_RUNG
   RUNG wire#w2
      Move(in := 2, out1 => #statCmdNummber)
   END_RUNG
   RUNG wire#w2
      Move(in := #tempAlignTableAxisXPosition, out1 => #statCmdParameter1)
   END_RUNG
   RUNG wire#w2
      Move(in := #tempAlignTableAxisY1Position, out1 => #statCmdParameter2)
   END_RUNG
   RUNG wire#w2
      Move(in := #tempAlignTableAxisY2Position, out1 => #statCmdParameter3)
   END_RUNG
   // the same network as SCL:
   #_w1 := #statAllMoveSeq = 20;
   IF #_w1 THEN
       #instAlignTableAxisXMCMoveAbs.Position := #statAxisXMovePosition[2];
       #instAlignTableAxisY1MCMoveAbs.Position := #statAxisY1MovePosition[2];
       #instAlignTableAxisY2MCMoveAbs.Position := #statAxisY2MovePosition[2];
   END_IF;
   #statMoveXCmd[2] := #_w1;
   #statMoveY1Cmd[2] := #_w1;
   #statMoveY2Cmd[2] := #_w1;
   #_w2 := #_w1 AND #instAlignTableAxisXMCMoveAbs.Done AND #instAlignTableAxisY1MCMoveAbs.Done AND #instAlignTableAxisY2MCMoveAbs.Done;
   #statTimer[3].TON(IN := #_w2, PT := #VISION_DELAY_TIME);
   IF #statTimer[3].Q THEN #statAllMoveSeq := 25; END_IF;
   IF #_w2 THEN
       #statCmdNummber := 2;
       #statCmdParameter1 := #tempAlignTableAxisXPosition;
       #statCmdParameter2 := #tempAlignTableAxisY1Position;
       #statCmdParameter3 := #tempAlignTableAxisY2Position;
   END_IF;
END_REGION

REGION Network 11: All Move Seq Pos 2 Vision Trigger [Seq 25]
   RUNG wire#powerrail
      { S7_Templates := "SrcType := DInt" } EQ_Contact(in1 := #statAllMoveSeq, in2 := 25)
      wire#w1
      Coil( #statRequstCmd[2] )
   END_RUNG
   RUNG wire#w1
      Contact( #statRequstCmd[2] )
      { S7_Templates := "time_type := Time" } #statTimer[34].TON(pt := #REQ_DELAY_TIME, et =>)
      Coil( #statVisionCmd[2] )
   END_RUNG
   RUNG wire#w1
      Contact( #statVisionCmd[2] )
      { S7_Templates := "time_type := Time" } #statTimer[4].TON(pt := #VISION_DELAY_TIME, et =>)
      Move(in := 27, out1 => #statAllMoveSeq)
   END_RUNG
   // the same network as SCL:
   #statRequstCmd[2] := #statAllMoveSeq = 25;
   #statTimer[34].TON(IN := (#statAllMoveSeq = 25) AND #statRequstCmd[2], PT := #REQ_DELAY_TIME);
   #statVisionCmd[2] := #statTimer[34].Q;
   #statTimer[4].TON(IN := (#statAllMoveSeq = 25) AND #statVisionCmd[2], PT := #VISION_DELAY_TIME);
   IF #statTimer[4].Q THEN #statAllMoveSeq := 27; END_IF;
END_REGION

REGION Network 12: All Move Seq Pos 2 Wait Cmd Complete Bit [Seq 27]
   RUNG wire#powerrail
      { S7_Templates := "SrcType := DInt" } EQ_Contact(in1 := #statAllMoveSeq, in2 := 27)
      wire#w1
      Coil( #statRequstCmd[12] )
   END_RUNG
   RUNG wire#w1
      Contact( #cmdComplete )
      Move(in := 30, out1 => #statAllMoveSeq)
   END_RUNG
   // the same network as SCL:
   #statRequstCmd[12] := #statAllMoveSeq = 27;
   IF (#statAllMoveSeq = 27) AND #cmdComplete THEN #statAllMoveSeq := 30; END_IF;
END_REGION

REGION Network 13: All Move Seq Pos 3 [Seq 30]
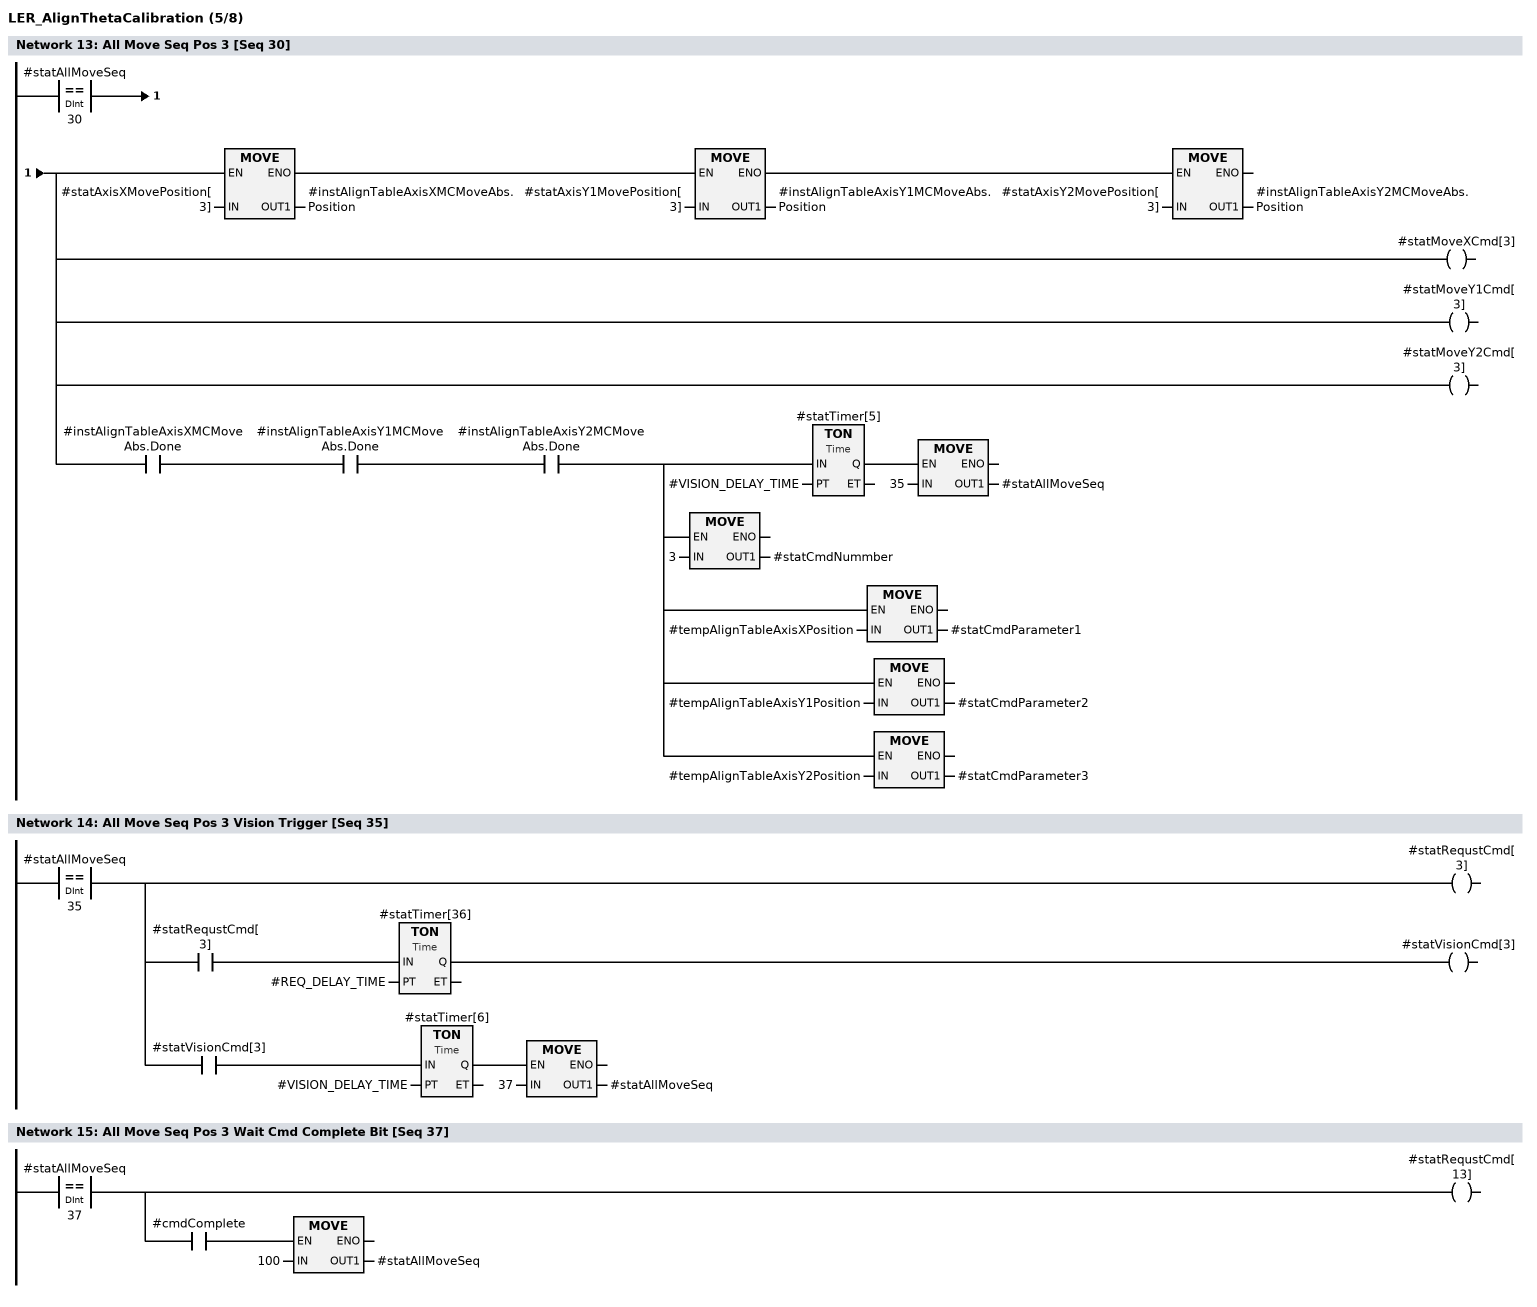
   RUNG wire#powerrail
      { S7_Templates := "SrcType := DInt" } EQ_Contact(in1 := #statAllMoveSeq, in2 := 30)
      wire#w1
      Move(in := #statAxisXMovePosition[3], out1 => #instAlignTableAxisXMCMoveAbs.Position)
      Move(in := #statAxisY1MovePosition[3], out1 => #instAlignTableAxisY1MCMoveAbs.Position)
      Move(in := #statAxisY2MovePosition[3], out1 => #instAlignTableAxisY2MCMoveAbs.Position)
   END_RUNG
   RUNG wire#w1
      Coil( #statMoveXCmd[3] )
   END_RUNG
   RUNG wire#w1
      Coil( #statMoveY1Cmd[3] )
   END_RUNG
   RUNG wire#w1
      Coil( #statMoveY2Cmd[3] )
   END_RUNG
   RUNG wire#w1
      Contact( #instAlignTableAxisXMCMoveAbs.Done )
      Contact( #instAlignTableAxisY1MCMoveAbs.Done )
      Contact( #instAlignTableAxisY2MCMoveAbs.Done )
      wire#w2
      { S7_Templates := "time_type := Time" } #statTimer[5].TON(pt := #VISION_DELAY_TIME, et =>)
      Move(in := 35, out1 => #statAllMoveSeq)
   END_RUNG
   RUNG wire#w2
      Move(in := 3, out1 => #statCmdNummber)
   END_RUNG
   RUNG wire#w2
      Move(in := #tempAlignTableAxisXPosition, out1 => #statCmdParameter1)
   END_RUNG
   RUNG wire#w2
      Move(in := #tempAlignTableAxisY1Position, out1 => #statCmdParameter2)
   END_RUNG
   RUNG wire#w2
      Move(in := #tempAlignTableAxisY2Position, out1 => #statCmdParameter3)
   END_RUNG
   // the same network as SCL:
   #_w1 := #statAllMoveSeq = 30;
   IF #_w1 THEN
       #instAlignTableAxisXMCMoveAbs.Position := #statAxisXMovePosition[3];
       #instAlignTableAxisY1MCMoveAbs.Position := #statAxisY1MovePosition[3];
       #instAlignTableAxisY2MCMoveAbs.Position := #statAxisY2MovePosition[3];
   END_IF;
   #statMoveXCmd[3] := #_w1;
   #statMoveY1Cmd[3] := #_w1;
   #statMoveY2Cmd[3] := #_w1;
   #_w2 := #_w1 AND #instAlignTableAxisXMCMoveAbs.Done AND #instAlignTableAxisY1MCMoveAbs.Done AND #instAlignTableAxisY2MCMoveAbs.Done;
   #statTimer[5].TON(IN := #_w2, PT := #VISION_DELAY_TIME);
   IF #statTimer[5].Q THEN #statAllMoveSeq := 35; END_IF;
   IF #_w2 THEN
       #statCmdNummber := 3;
       #statCmdParameter1 := #tempAlignTableAxisXPosition;
       #statCmdParameter2 := #tempAlignTableAxisY1Position;
       #statCmdParameter3 := #tempAlignTableAxisY2Position;
   END_IF;
END_REGION

REGION Network 14: All Move Seq Pos 3 Vision Trigger [Seq 35]
   RUNG wire#powerrail
      { S7_Templates := "SrcType := DInt" } EQ_Contact(in1 := #statAllMoveSeq, in2 := 35)
      wire#w1
      Coil( #statRequstCmd[3] )
   END_RUNG
   RUNG wire#w1
      Contact( #statRequstCmd[3] )
      { S7_Templates := "time_type := Time" } #statTimer[36].TON(pt := #REQ_DELAY_TIME, et =>)
      Coil( #statVisionCmd[3] )
   END_RUNG
   RUNG wire#w1
      Contact( #statVisionCmd[3] )
      { S7_Templates := "time_type := Time" } #statTimer[6].TON(pt := #VISION_DELAY_TIME, et =>)
      Move(in := 37, out1 => #statAllMoveSeq)
   END_RUNG
   // the same network as SCL:
   #statRequstCmd[3] := #statAllMoveSeq = 35;
   #statTimer[36].TON(IN := (#statAllMoveSeq = 35) AND #statRequstCmd[3], PT := #REQ_DELAY_TIME);
   #statVisionCmd[3] := #statTimer[36].Q;
   #statTimer[6].TON(IN := (#statAllMoveSeq = 35) AND #statVisionCmd[3], PT := #VISION_DELAY_TIME);
   IF #statTimer[6].Q THEN #statAllMoveSeq := 37; END_IF;
END_REGION

REGION Network 15: All Move Seq Pos 3 Wait Cmd Complete Bit [Seq 37]
   RUNG wire#powerrail
      { S7_Templates := "SrcType := DInt" } EQ_Contact(in1 := #statAllMoveSeq, in2 := 37)
      wire#w1
      Coil( #statRequstCmd[13] )
   END_RUNG
   RUNG wire#w1
      Contact( #cmdComplete )
      Move(in := 100, out1 => #statAllMoveSeq)
   END_RUNG
   // the same network as SCL:
   #statRequstCmd[13] := #statAllMoveSeq = 37;
   IF (#statAllMoveSeq = 37) AND #cmdComplete THEN #statAllMoveSeq := 100; END_IF;
END_REGION

REGION Network 16: All Move Seq Done [Seq 100]
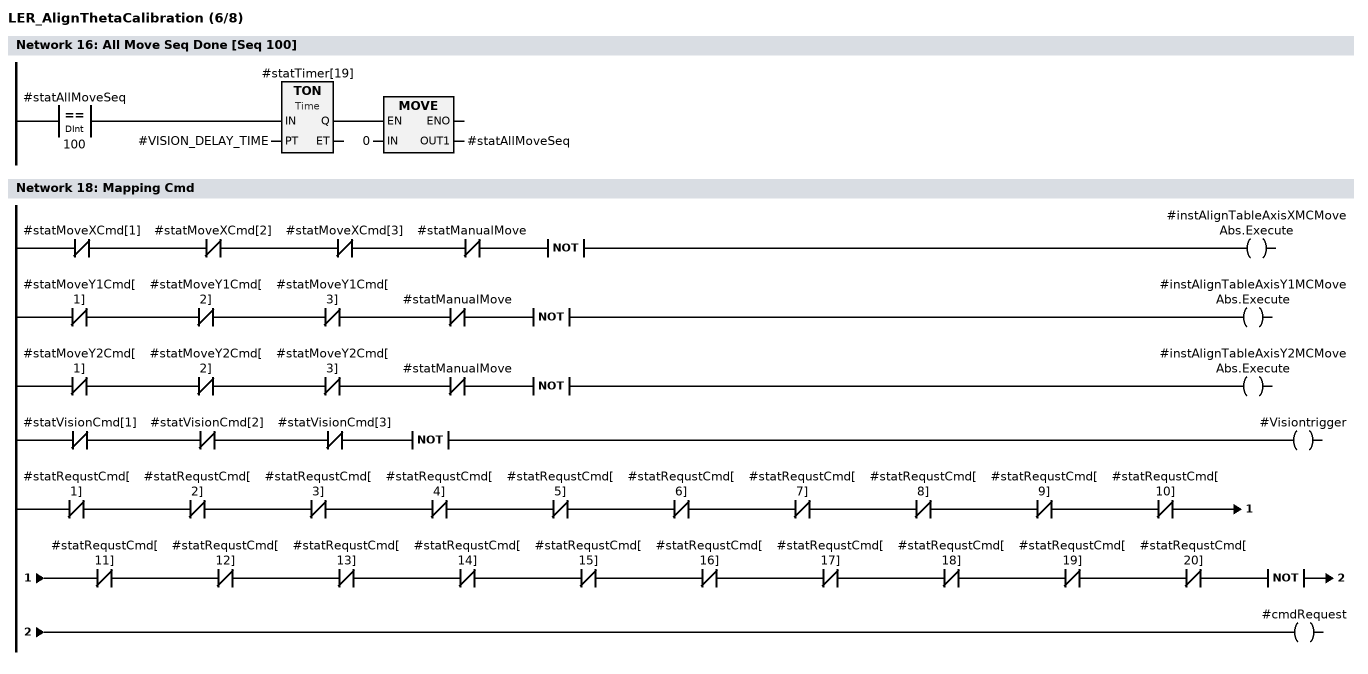
   RUNG wire#powerrail
      { S7_Templates := "SrcType := DInt" } EQ_Contact(in1 := #statAllMoveSeq, in2 := 100)
      { S7_Templates := "time_type := Time" } #statTimer[19].TON(pt := #VISION_DELAY_TIME, et =>)
      Move(in := 0, out1 => #statAllMoveSeq)
   END_RUNG
   // the same network as SCL:
   #statTimer[19].TON(IN := #statAllMoveSeq = 100, PT := #VISION_DELAY_TIME);
   IF #statTimer[19].Q THEN #statAllMoveSeq := 0; END_IF;
END_REGION

REGION Network 17: === Sequence End ===
END_REGION

REGION Network 18: Mapping Cmd
   RUNG wire#powerrail
      I_Contact( #statMoveXCmd[1] )
      I_Contact( #statMoveXCmd[2] )
      I_Contact( #statMoveXCmd[3] )
      I_Contact( #statManualMove )
      Not()
      Coil( #instAlignTableAxisXMCMoveAbs.Execute )
   END_RUNG
   RUNG wire#powerrail
      I_Contact( #statMoveY1Cmd[1] )
      I_Contact( #statMoveY1Cmd[2] )
      I_Contact( #statMoveY1Cmd[3] )
      I_Contact( #statManualMove )
      Not()
      Coil( #instAlignTableAxisY1MCMoveAbs.Execute )
   END_RUNG
   RUNG wire#powerrail
      I_Contact( #statMoveY2Cmd[1] )
      I_Contact( #statMoveY2Cmd[2] )
      I_Contact( #statMoveY2Cmd[3] )
      I_Contact( #statManualMove )
      Not()
      Coil( #instAlignTableAxisY2MCMoveAbs.Execute )
   END_RUNG
   RUNG wire#powerrail
      I_Contact( #statVisionCmd[1] )
      I_Contact( #statVisionCmd[2] )
      I_Contact( #statVisionCmd[3] )
      Not()
      Coil( #Visiontrigger )
   END_RUNG
   RUNG wire#powerrail
      I_Contact( #statRequstCmd[1] )
      I_Contact( #statRequstCmd[2] )
      I_Contact( #statRequstCmd[3] )
      I_Contact( #statRequstCmd[4] )
      I_Contact( #statRequstCmd[5] )
      I_Contact( #statRequstCmd[6] )
      I_Contact( #statRequstCmd[7] )
      I_Contact( #statRequstCmd[8] )
      I_Contact( #statRequstCmd[9] )
      I_Contact( #statRequstCmd[10] )
      I_Contact( #statRequstCmd[11] )
      I_Contact( #statRequstCmd[12] )
      I_Contact( #statRequstCmd[13] )
      I_Contact( #statRequstCmd[14] )
      I_Contact( #statRequstCmd[15] )
      I_Contact( #statRequstCmd[16] )
      I_Contact( #statRequstCmd[17] )
      I_Contact( #statRequstCmd[18] )
      I_Contact( #statRequstCmd[19] )
      I_Contact( #statRequstCmd[20] )
      Not()
      Coil( #cmdRequest )
   END_RUNG
   // the same network as SCL:
   #instAlignTableAxisXMCMoveAbs.Execute := NOT (NOT #statMoveXCmd[1] AND NOT #statMoveXCmd[2] AND NOT #statMoveXCmd[3] AND NOT #statManualMove);
   #instAlignTableAxisY1MCMoveAbs.Execute := NOT (NOT #statMoveY1Cmd[1] AND NOT #statMoveY1Cmd[2] AND NOT #statMoveY1Cmd[3] AND NOT #statManualMove);
   #instAlignTableAxisY2MCMoveAbs.Execute := NOT (NOT #statMoveY2Cmd[1] AND NOT #statMoveY2Cmd[2] AND NOT #statMoveY2Cmd[3] AND NOT #statManualMove);
   #Visiontrigger := NOT (NOT #statVisionCmd[1] AND NOT #statVisionCmd[2] AND NOT #statVisionCmd[3]);
   #cmdRequest := NOT (NOT #statRequstCmd[1] AND NOT #statRequstCmd[2] AND NOT #statRequstCmd[3] AND NOT #statRequstCmd[4] AND NOT #statRequstCmd[5] AND NOT #statRequstCmd[6] AND NOT #statRequstCmd[7] AND NOT #statRequstCmd[8] AND NOT #statRequstCmd[9] AND NOT #statRequstCmd[10] AND NOT #statRequstCmd[11] AND NOT #statRequstCmd[12] AND NOT #statRequstCmd[13] AND NOT #statRequstCmd[14] AND NOT #statRequstCmd[15] AND NOT #statRequstCmd[16] AND NOT #statRequstCmd[17] AND NOT #statRequstCmd[18] AND NOT #statRequstCmd[19] AND NOT #statRequstCmd[20]);
END_REGION

REGION Network 19: Call Instance
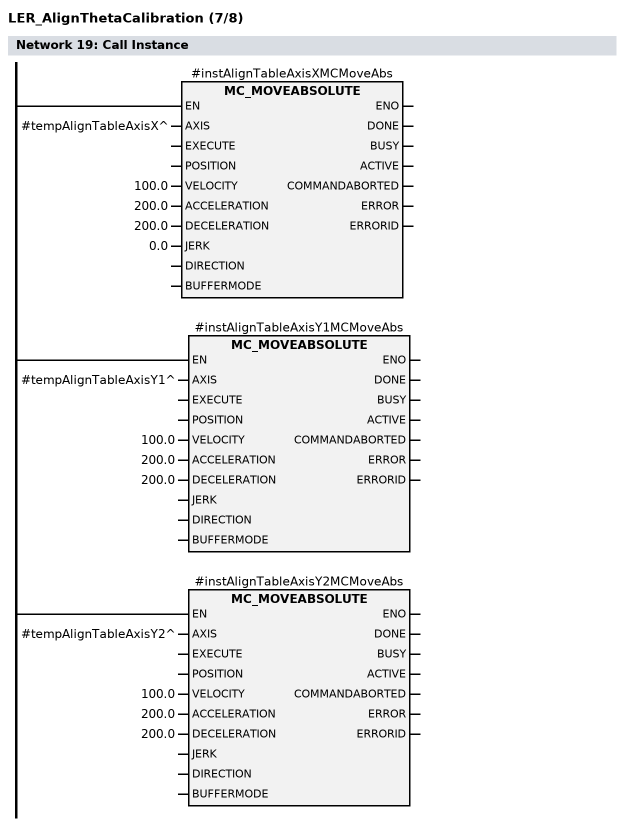
   RUNG wire#powerrail
      #instAlignTableAxisXMCMoveAbs.MC_MOVEABSOLUTE(Axis := #tempAlignTableAxisX^, Execute :=, Position :=, Velocity := 100.0, Acceleration := 200.0, Deceleration := 200.0, Jerk := 0.0, Direction :=, BufferMode :=, Done =>, Busy =>, Active =>, CommandAborted =>, Error =>, ErrorId =>)
   END_RUNG
   RUNG wire#powerrail
      #instAlignTableAxisY1MCMoveAbs.MC_MOVEABSOLUTE(Axis := #tempAlignTableAxisY1^, Execute :=, Position :=, Velocity := 100.0, Acceleration := 200.0, Deceleration := 200.0, Jerk :=, Direction :=, BufferMode :=, Done =>, Busy =>, Active =>, CommandAborted =>, Error =>, ErrorId =>)
   END_RUNG
   RUNG wire#powerrail
      #instAlignTableAxisY2MCMoveAbs.MC_MOVEABSOLUTE(Axis := #tempAlignTableAxisY2^, Execute :=, Position :=, Velocity := 100.0, Acceleration := 200.0, Deceleration := 200.0, Jerk :=, Direction :=, BufferMode :=, Done =>, Busy =>, Active =>, CommandAborted =>, Error =>, ErrorId =>)
   END_RUNG
   // the same network as SCL:
   #instAlignTableAxisXMCMoveAbs(Axis := #tempAlignTableAxisX^,   // MC_MOVEABSOLUTE
                           Velocity := 100.0,
                           Acceleration := 200.0,
                           Deceleration := 200.0,
                           Jerk := 0.0);
   #instAlignTableAxisY1MCMoveAbs(Axis := #tempAlignTableAxisY1^,   // MC_MOVEABSOLUTE
                           Velocity := 100.0,
                           Acceleration := 200.0,
                           Deceleration := 200.0);
   #instAlignTableAxisY2MCMoveAbs(Axis := #tempAlignTableAxisY2^,   // MC_MOVEABSOLUTE
                           Velocity := 100.0,
                           Acceleration := 200.0,
                           Deceleration := 200.0);
END_REGION

REGION Network 20: Mapping Output
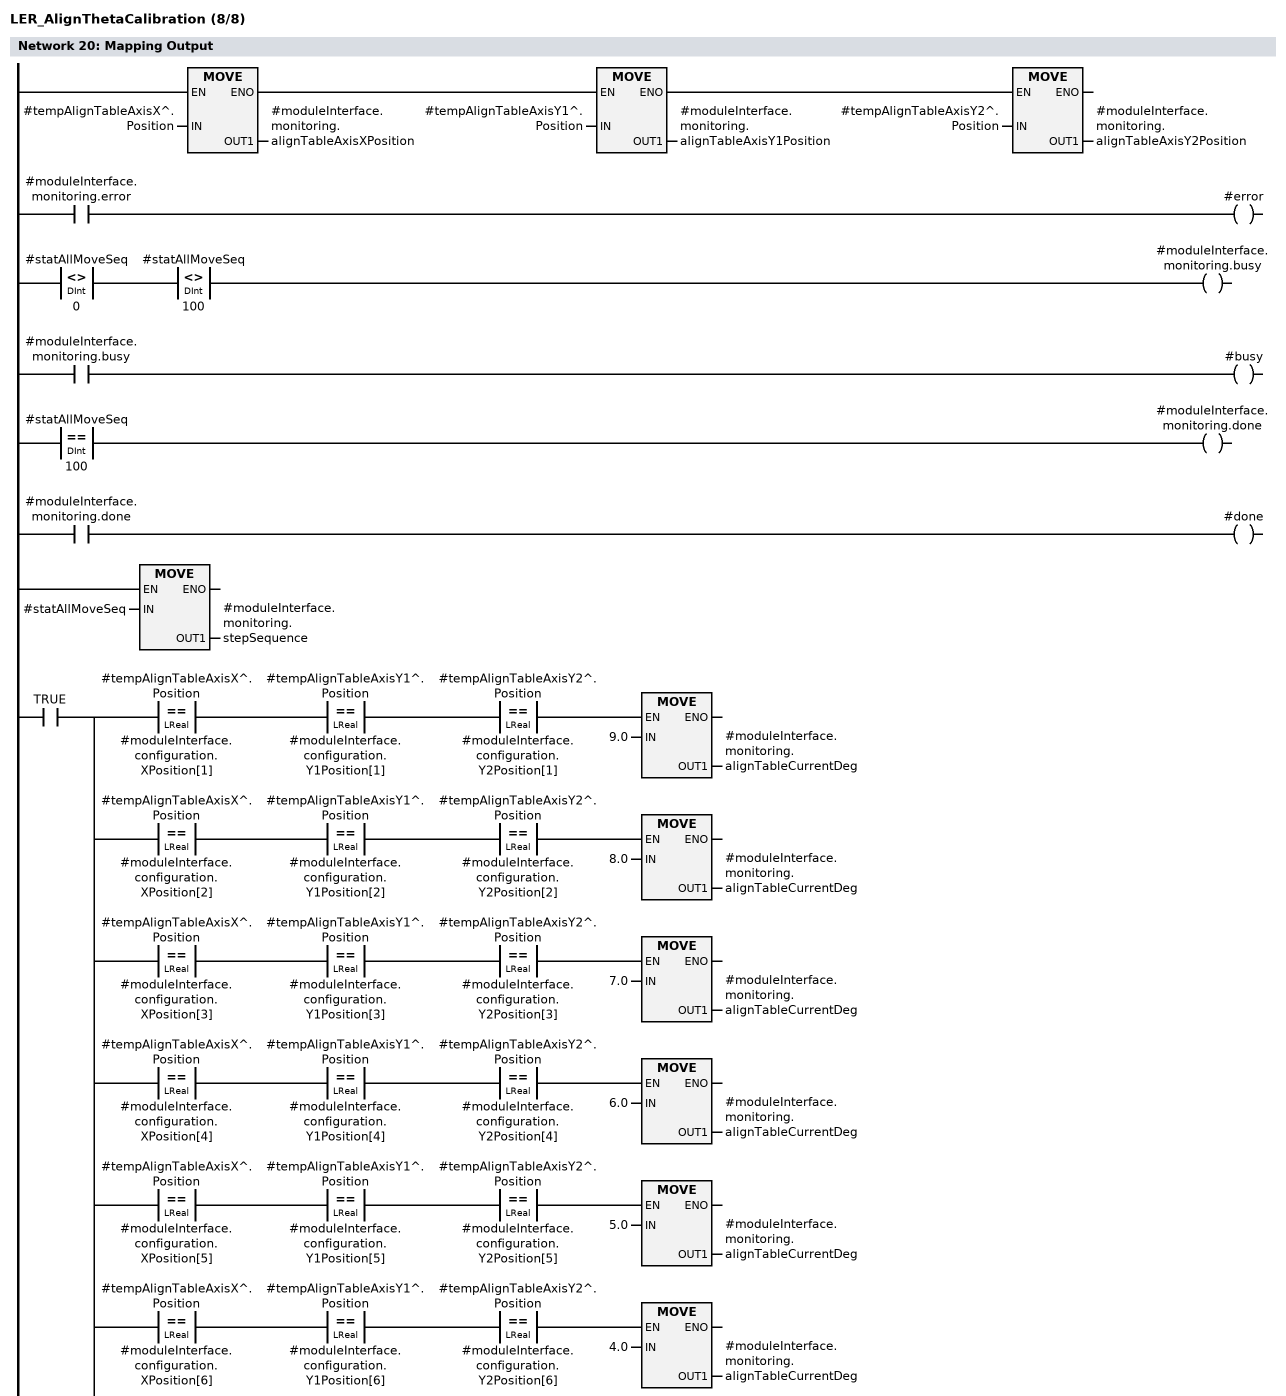
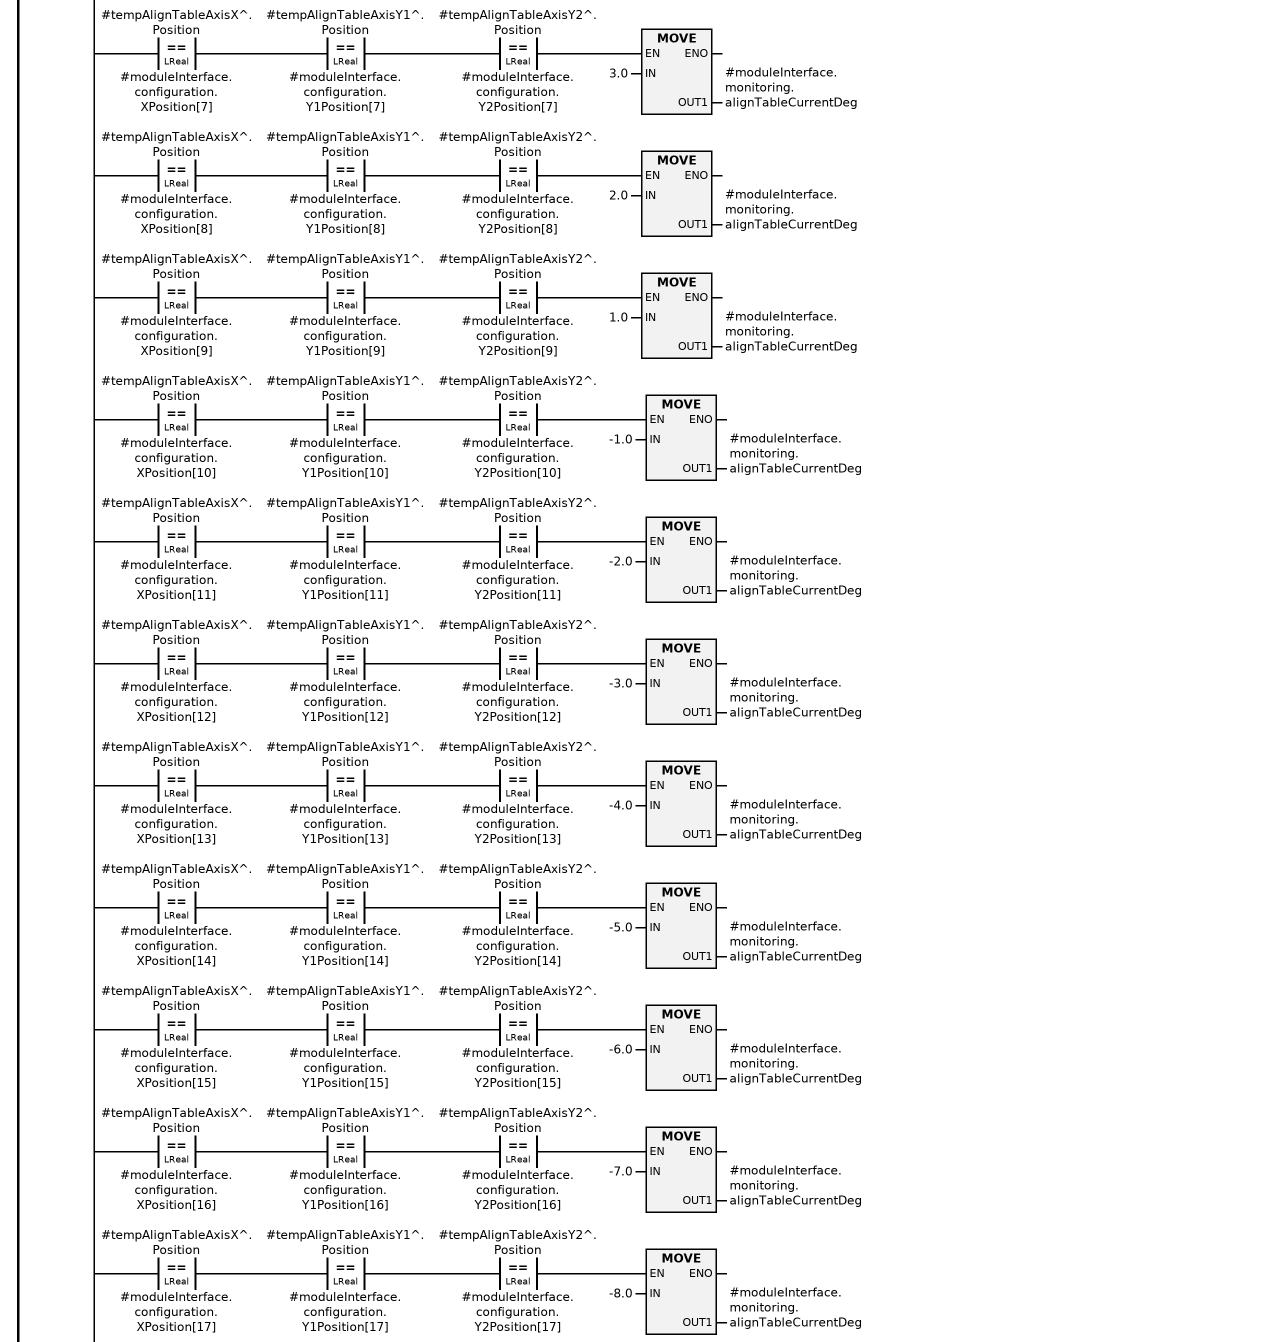
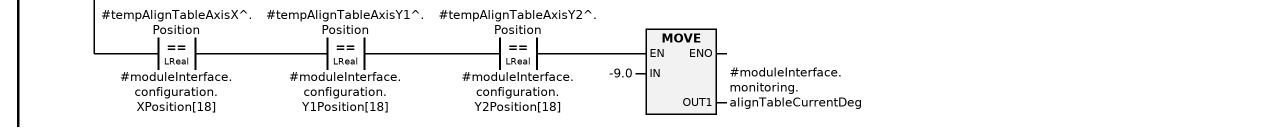
   RUNG wire#powerrail
      Move(in := #tempAlignTableAxisX^.Position, out1 => #moduleInterface.monitoring.alignTableAxisXPosition)
      Move(in := #tempAlignTableAxisY1^.Position, out1 => #moduleInterface.monitoring.alignTableAxisY1Position)
      Move(in := #tempAlignTableAxisY2^.Position, out1 => #moduleInterface.monitoring.alignTableAxisY2Position)
   END_RUNG
   RUNG wire#powerrail
      Contact( #moduleInterface.monitoring.error )
      Coil( #error )
   END_RUNG
   RUNG wire#powerrail
      { S7_Templates := "SrcType := DInt" } NE_Contact(in1 := #statAllMoveSeq, in2 := 0)
      { S7_Templates := "SrcType := DInt" } NE_Contact(in1 := #statAllMoveSeq, in2 := 100)
      Coil( #moduleInterface.monitoring.busy )
   END_RUNG
   RUNG wire#powerrail
      Contact( #moduleInterface.monitoring.busy )
      Coil( #busy )
   END_RUNG
   RUNG wire#powerrail
      { S7_Templates := "SrcType := DInt" } EQ_Contact(in1 := #statAllMoveSeq, in2 := 100)
      Coil( #moduleInterface.monitoring.done )
   END_RUNG
   RUNG wire#powerrail
      Contact( #moduleInterface.monitoring.done )
      Coil( #done )
   END_RUNG
   RUNG wire#powerrail
      Move(in := #statAllMoveSeq, out1 => #moduleInterface.monitoring.stepSequence)
   END_RUNG
   RUNG wire#powerrail
      Contact( TRUE )
      wire#w1
      { S7_Templates := "SrcType := LReal" } EQ_Contact(in1 := #tempAlignTableAxisX^.Position, in2 := #moduleInterface.configuration.XPosition[1])
      { S7_Templates := "SrcType := LReal" } EQ_Contact(in1 := #tempAlignTableAxisY1^.Position, in2 := #moduleInterface.configuration.Y1Position[1])
      { S7_Templates := "SrcType := LReal" } EQ_Contact(in1 := #tempAlignTableAxisY2^.Position, in2 := #moduleInterface.configuration.Y2Position[1])
      Move(in := 9.0, out1 => #moduleInterface.monitoring.alignTableCurrentDeg)
   END_RUNG
   RUNG wire#w1
      { S7_Templates := "SrcType := LReal" } EQ_Contact(in1 := #tempAlignTableAxisX^.Position, in2 := #moduleInterface.configuration.XPosition[2])
      { S7_Templates := "SrcType := LReal" } EQ_Contact(in1 := #tempAlignTableAxisY1^.Position, in2 := #moduleInterface.configuration.Y1Position[2])
      { S7_Templates := "SrcType := LReal" } EQ_Contact(in1 := #tempAlignTableAxisY2^.Position, in2 := #moduleInterface.configuration.Y2Position[2])
      Move(in := 8.0, out1 => #moduleInterface.monitoring.alignTableCurrentDeg)
   END_RUNG
   RUNG wire#w1
      { S7_Templates := "SrcType := LReal" } EQ_Contact(in1 := #tempAlignTableAxisX^.Position, in2 := #moduleInterface.configuration.XPosition[3])
      { S7_Templates := "SrcType := LReal" } EQ_Contact(in1 := #tempAlignTableAxisY1^.Position, in2 := #moduleInterface.configuration.Y1Position[3])
      { S7_Templates := "SrcType := LReal" } EQ_Contact(in1 := #tempAlignTableAxisY2^.Position, in2 := #moduleInterface.configuration.Y2Position[3])
      Move(in := 7.0, out1 => #moduleInterface.monitoring.alignTableCurrentDeg)
   END_RUNG
   RUNG wire#w1
      { S7_Templates := "SrcType := LReal" } EQ_Contact(in1 := #tempAlignTableAxisX^.Position, in2 := #moduleInterface.configuration.XPosition[4])
      { S7_Templates := "SrcType := LReal" } EQ_Contact(in1 := #tempAlignTableAxisY1^.Position, in2 := #moduleInterface.configuration.Y1Position[4])
      { S7_Templates := "SrcType := LReal" } EQ_Contact(in1 := #tempAlignTableAxisY2^.Position, in2 := #moduleInterface.configuration.Y2Position[4])
      Move(in := 6.0, out1 => #moduleInterface.monitoring.alignTableCurrentDeg)
   END_RUNG
   RUNG wire#w1
      { S7_Templates := "SrcType := LReal" } EQ_Contact(in1 := #tempAlignTableAxisX^.Position, in2 := #moduleInterface.configuration.XPosition[5])
      { S7_Templates := "SrcType := LReal" } EQ_Contact(in1 := #tempAlignTableAxisY1^.Position, in2 := #moduleInterface.configuration.Y1Position[5])
      { S7_Templates := "SrcType := LReal" } EQ_Contact(in1 := #tempAlignTableAxisY2^.Position, in2 := #moduleInterface.configuration.Y2Position[5])
      Move(in := 5.0, out1 => #moduleInterface.monitoring.alignTableCurrentDeg)
   END_RUNG
   RUNG wire#w1
      { S7_Templates := "SrcType := LReal" } EQ_Contact(in1 := #tempAlignTableAxisX^.Position, in2 := #moduleInterface.configuration.XPosition[6])
      { S7_Templates := "SrcType := LReal" } EQ_Contact(in1 := #tempAlignTableAxisY1^.Position, in2 := #moduleInterface.configuration.Y1Position[6])
      { S7_Templates := "SrcType := LReal" } EQ_Contact(in1 := #tempAlignTableAxisY2^.Position, in2 := #moduleInterface.configuration.Y2Position[6])
      Move(in := 4.0, out1 => #moduleInterface.monitoring.alignTableCurrentDeg)
   END_RUNG
   RUNG wire#w1
      { S7_Templates := "SrcType := LReal" } EQ_Contact(in1 := #tempAlignTableAxisX^.Position, in2 := #moduleInterface.configuration.XPosition[7])
      { S7_Templates := "SrcType := LReal" } EQ_Contact(in1 := #tempAlignTableAxisY1^.Position, in2 := #moduleInterface.configuration.Y1Position[7])
      { S7_Templates := "SrcType := LReal" } EQ_Contact(in1 := #tempAlignTableAxisY2^.Position, in2 := #moduleInterface.configuration.Y2Position[7])
      Move(in := 3.0, out1 => #moduleInterface.monitoring.alignTableCurrentDeg)
   END_RUNG
   RUNG wire#w1
      { S7_Templates := "SrcType := LReal" } EQ_Contact(in1 := #tempAlignTableAxisX^.Position, in2 := #moduleInterface.configuration.XPosition[8])
      { S7_Templates := "SrcType := LReal" } EQ_Contact(in1 := #tempAlignTableAxisY1^.Position, in2 := #moduleInterface.configuration.Y1Position[8])
      { S7_Templates := "SrcType := LReal" } EQ_Contact(in1 := #tempAlignTableAxisY2^.Position, in2 := #moduleInterface.configuration.Y2Position[8])
      Move(in := 2.0, out1 => #moduleInterface.monitoring.alignTableCurrentDeg)
   END_RUNG
   RUNG wire#w1
      { S7_Templates := "SrcType := LReal" } EQ_Contact(in1 := #tempAlignTableAxisX^.Position, in2 := #moduleInterface.configuration.XPosition[9])
      { S7_Templates := "SrcType := LReal" } EQ_Contact(in1 := #tempAlignTableAxisY1^.Position, in2 := #moduleInterface.configuration.Y1Position[9])
      { S7_Templates := "SrcType := LReal" } EQ_Contact(in1 := #tempAlignTableAxisY2^.Position, in2 := #moduleInterface.configuration.Y2Position[9])
      Move(in := 1.0, out1 => #moduleInterface.monitoring.alignTableCurrentDeg)
   END_RUNG
   RUNG wire#w1
      { S7_Templates := "SrcType := LReal" } EQ_Contact(in1 := #tempAlignTableAxisX^.Position, in2 := #moduleInterface.configuration.XPosition[10])
      { S7_Templates := "SrcType := LReal" } EQ_Contact(in1 := #tempAlignTableAxisY1^.Position, in2 := #moduleInterface.configuration.Y1Position[10])
      { S7_Templates := "SrcType := LReal" } EQ_Contact(in1 := #tempAlignTableAxisY2^.Position, in2 := #moduleInterface.configuration.Y2Position[10])
      Move(in := -1.0, out1 => #moduleInterface.monitoring.alignTableCurrentDeg)
   END_RUNG
   RUNG wire#w1
      { S7_Templates := "SrcType := LReal" } EQ_Contact(in1 := #tempAlignTableAxisX^.Position, in2 := #moduleInterface.configuration.XPosition[11])
      { S7_Templates := "SrcType := LReal" } EQ_Contact(in1 := #tempAlignTableAxisY1^.Position, in2 := #moduleInterface.configuration.Y1Position[11])
      { S7_Templates := "SrcType := LReal" } EQ_Contact(in1 := #tempAlignTableAxisY2^.Position, in2 := #moduleInterface.configuration.Y2Position[11])
      Move(in := -2.0, out1 => #moduleInterface.monitoring.alignTableCurrentDeg)
   END_RUNG
   RUNG wire#w1
      { S7_Templates := "SrcType := LReal" } EQ_Contact(in1 := #tempAlignTableAxisX^.Position, in2 := #moduleInterface.configuration.XPosition[12])
      { S7_Templates := "SrcType := LReal" } EQ_Contact(in1 := #tempAlignTableAxisY1^.Position, in2 := #moduleInterface.configuration.Y1Position[12])
      { S7_Templates := "SrcType := LReal" } EQ_Contact(in1 := #tempAlignTableAxisY2^.Position, in2 := #moduleInterface.configuration.Y2Position[12])
      Move(in := -3.0, out1 => #moduleInterface.monitoring.alignTableCurrentDeg)
   END_RUNG
   RUNG wire#w1
      { S7_Templates := "SrcType := LReal" } EQ_Contact(in1 := #tempAlignTableAxisX^.Position, in2 := #moduleInterface.configuration.XPosition[13])
      { S7_Templates := "SrcType := LReal" } EQ_Contact(in1 := #tempAlignTableAxisY1^.Position, in2 := #moduleInterface.configuration.Y1Position[13])
      { S7_Templates := "SrcType := LReal" } EQ_Contact(in1 := #tempAlignTableAxisY2^.Position, in2 := #moduleInterface.configuration.Y2Position[13])
      Move(in := -4.0, out1 => #moduleInterface.monitoring.alignTableCurrentDeg)
   END_RUNG
   RUNG wire#w1
      { S7_Templates := "SrcType := LReal" } EQ_Contact(in1 := #tempAlignTableAxisX^.Position, in2 := #moduleInterface.configuration.XPosition[14])
      { S7_Templates := "SrcType := LReal" } EQ_Contact(in1 := #tempAlignTableAxisY1^.Position, in2 := #moduleInterface.configuration.Y1Position[14])
      { S7_Templates := "SrcType := LReal" } EQ_Contact(in1 := #tempAlignTableAxisY2^.Position, in2 := #moduleInterface.configuration.Y2Position[14])
      Move(in := -5.0, out1 => #moduleInterface.monitoring.alignTableCurrentDeg)
   END_RUNG
   RUNG wire#w1
      { S7_Templates := "SrcType := LReal" } EQ_Contact(in1 := #tempAlignTableAxisX^.Position, in2 := #moduleInterface.configuration.XPosition[15])
      { S7_Templates := "SrcType := LReal" } EQ_Contact(in1 := #tempAlignTableAxisY1^.Position, in2 := #moduleInterface.configuration.Y1Position[15])
      { S7_Templates := "SrcType := LReal" } EQ_Contact(in1 := #tempAlignTableAxisY2^.Position, in2 := #moduleInterface.configuration.Y2Position[15])
      Move(in := -6.0, out1 => #moduleInterface.monitoring.alignTableCurrentDeg)
   END_RUNG
   RUNG wire#w1
      { S7_Templates := "SrcType := LReal" } EQ_Contact(in1 := #tempAlignTableAxisX^.Position, in2 := #moduleInterface.configuration.XPosition[16])
      { S7_Templates := "SrcType := LReal" } EQ_Contact(in1 := #tempAlignTableAxisY1^.Position, in2 := #moduleInterface.configuration.Y1Position[16])
      { S7_Templates := "SrcType := LReal" } EQ_Contact(in1 := #tempAlignTableAxisY2^.Position, in2 := #moduleInterface.configuration.Y2Position[16])
      Move(in := -7.0, out1 => #moduleInterface.monitoring.alignTableCurrentDeg)
   END_RUNG
   RUNG wire#w1
      { S7_Templates := "SrcType := LReal" } EQ_Contact(in1 := #tempAlignTableAxisX^.Position, in2 := #moduleInterface.configuration.XPosition[17])
      { S7_Templates := "SrcType := LReal" } EQ_Contact(in1 := #tempAlignTableAxisY1^.Position, in2 := #moduleInterface.configuration.Y1Position[17])
      { S7_Templates := "SrcType := LReal" } EQ_Contact(in1 := #tempAlignTableAxisY2^.Position, in2 := #moduleInterface.configuration.Y2Position[17])
      Move(in := -8.0, out1 => #moduleInterface.monitoring.alignTableCurrentDeg)
   END_RUNG
   RUNG wire#w1
      { S7_Templates := "SrcType := LReal" } EQ_Contact(in1 := #tempAlignTableAxisX^.Position, in2 := #moduleInterface.configuration.XPosition[18])
      { S7_Templates := "SrcType := LReal" } EQ_Contact(in1 := #tempAlignTableAxisY1^.Position, in2 := #moduleInterface.configuration.Y1Position[18])
      { S7_Templates := "SrcType := LReal" } EQ_Contact(in1 := #tempAlignTableAxisY2^.Position, in2 := #moduleInterface.configuration.Y2Position[18])
      Move(in := -9.0, out1 => #moduleInterface.monitoring.alignTableCurrentDeg)
   END_RUNG
   // the same network as SCL:
   #moduleInterface.monitoring.alignTableAxisXPosition := #tempAlignTableAxisX^.Position;
   #moduleInterface.monitoring.alignTableAxisY1Position := #tempAlignTableAxisY1^.Position;
   #moduleInterface.monitoring.alignTableAxisY2Position := #tempAlignTableAxisY2^.Position;
   #error := #moduleInterface.monitoring.error;
   #moduleInterface.monitoring.busy := (#statAllMoveSeq <> 0) AND (#statAllMoveSeq <> 100);
   #busy := #moduleInterface.monitoring.busy;
   #moduleInterface.monitoring.done := #statAllMoveSeq = 100;
   #done := #moduleInterface.monitoring.done;
   #moduleInterface.monitoring.stepSequence := #statAllMoveSeq;
   IF TRUE AND (#tempAlignTableAxisX^.Position = #moduleInterface.configuration.XPosition[1]) AND (#tempAlignTableAxisY1^.Position = #moduleInterface.configuration.Y1Position[1]) AND (#tempAlignTableAxisY2^.Position = #moduleInterface.configuration.Y2Position[1]) THEN
       #moduleInterface.monitoring.alignTableCurrentDeg := 9.0;
   END_IF;
   IF TRUE AND (#tempAlignTableAxisX^.Position = #moduleInterface.configuration.XPosition[2]) AND (#tempAlignTableAxisY1^.Position = #moduleInterface.configuration.Y1Position[2]) AND (#tempAlignTableAxisY2^.Position = #moduleInterface.configuration.Y2Position[2]) THEN
       #moduleInterface.monitoring.alignTableCurrentDeg := 8.0;
   END_IF;
   IF TRUE AND (#tempAlignTableAxisX^.Position = #moduleInterface.configuration.XPosition[3]) AND (#tempAlignTableAxisY1^.Position = #moduleInterface.configuration.Y1Position[3]) AND (#tempAlignTableAxisY2^.Position = #moduleInterface.configuration.Y2Position[3]) THEN
       #moduleInterface.monitoring.alignTableCurrentDeg := 7.0;
   END_IF;
   IF TRUE AND (#tempAlignTableAxisX^.Position = #moduleInterface.configuration.XPosition[4]) AND (#tempAlignTableAxisY1^.Position = #moduleInterface.configuration.Y1Position[4]) AND (#tempAlignTableAxisY2^.Position = #moduleInterface.configuration.Y2Position[4]) THEN
       #moduleInterface.monitoring.alignTableCurrentDeg := 6.0;
   END_IF;
   IF TRUE AND (#tempAlignTableAxisX^.Position = #moduleInterface.configuration.XPosition[5]) AND (#tempAlignTableAxisY1^.Position = #moduleInterface.configuration.Y1Position[5]) AND (#tempAlignTableAxisY2^.Position = #moduleInterface.configuration.Y2Position[5]) THEN
       #moduleInterface.monitoring.alignTableCurrentDeg := 5.0;
   END_IF;
   IF TRUE AND (#tempAlignTableAxisX^.Position = #moduleInterface.configuration.XPosition[6]) AND (#tempAlignTableAxisY1^.Position = #moduleInterface.configuration.Y1Position[6]) AND (#tempAlignTableAxisY2^.Position = #moduleInterface.configuration.Y2Position[6]) THEN
       #moduleInterface.monitoring.alignTableCurrentDeg := 4.0;
   END_IF;
   IF TRUE AND (#tempAlignTableAxisX^.Position = #moduleInterface.configuration.XPosition[7]) AND (#tempAlignTableAxisY1^.Position = #moduleInterface.configuration.Y1Position[7]) AND (#tempAlignTableAxisY2^.Position = #moduleInterface.configuration.Y2Position[7]) THEN
       #moduleInterface.monitoring.alignTableCurrentDeg := 3.0;
   END_IF;
   IF TRUE AND (#tempAlignTableAxisX^.Position = #moduleInterface.configuration.XPosition[8]) AND (#tempAlignTableAxisY1^.Position = #moduleInterface.configuration.Y1Position[8]) AND (#tempAlignTableAxisY2^.Position = #moduleInterface.configuration.Y2Position[8]) THEN
       #moduleInterface.monitoring.alignTableCurrentDeg := 2.0;
   END_IF;
   IF TRUE AND (#tempAlignTableAxisX^.Position = #moduleInterface.configuration.XPosition[9]) AND (#tempAlignTableAxisY1^.Position = #moduleInterface.configuration.Y1Position[9]) AND (#tempAlignTableAxisY2^.Position = #moduleInterface.configuration.Y2Position[9]) THEN
       #moduleInterface.monitoring.alignTableCurrentDeg := 1.0;
   END_IF;
   IF TRUE AND (#tempAlignTableAxisX^.Position = #moduleInterface.configuration.XPosition[10]) AND (#tempAlignTableAxisY1^.Position = #moduleInterface.configuration.Y1Position[10]) AND (#tempAlignTableAxisY2^.Position = #moduleInterface.configuration.Y2Position[10]) THEN
       #moduleInterface.monitoring.alignTableCurrentDeg := -1.0;
   END_IF;
   IF TRUE AND (#tempAlignTableAxisX^.Position = #moduleInterface.configuration.XPosition[11]) AND (#tempAlignTableAxisY1^.Position = #moduleInterface.configuration.Y1Position[11]) AND (#tempAlignTableAxisY2^.Position = #moduleInterface.configuration.Y2Position[11]) THEN
       #moduleInterface.monitoring.alignTableCurrentDeg := -2.0;
   END_IF;
   IF TRUE AND (#tempAlignTableAxisX^.Position = #moduleInterface.configuration.XPosition[12]) AND (#tempAlignTableAxisY1^.Position = #moduleInterface.configuration.Y1Position[12]) AND (#tempAlignTableAxisY2^.Position = #moduleInterface.configuration.Y2Position[12]) THEN
       #moduleInterface.monitoring.alignTableCurrentDeg := -3.0;
   END_IF;
   IF TRUE AND (#tempAlignTableAxisX^.Position = #moduleInterface.configuration.XPosition[13]) AND (#tempAlignTableAxisY1^.Position = #moduleInterface.configuration.Y1Position[13]) AND (#tempAlignTableAxisY2^.Position = #moduleInterface.configuration.Y2Position[13]) THEN
       #moduleInterface.monitoring.alignTableCurrentDeg := -4.0;
   END_IF;
   IF TRUE AND (#tempAlignTableAxisX^.Position = #moduleInterface.configuration.XPosition[14]) AND (#tempAlignTableAxisY1^.Position = #moduleInterface.configuration.Y1Position[14]) AND (#tempAlignTableAxisY2^.Position = #moduleInterface.configuration.Y2Position[14]) THEN
       #moduleInterface.monitoring.alignTableCurrentDeg := -5.0;
   END_IF;
   IF TRUE AND (#tempAlignTableAxisX^.Position = #moduleInterface.configuration.XPosition[15]) AND (#tempAlignTableAxisY1^.Position = #moduleInterface.configuration.Y1Position[15]) AND (#tempAlignTableAxisY2^.Position = #moduleInterface.configuration.Y2Position[15]) THEN
       #moduleInterface.monitoring.alignTableCurrentDeg := -6.0;
   END_IF;
   IF TRUE AND (#tempAlignTableAxisX^.Position = #moduleInterface.configuration.XPosition[16]) AND (#tempAlignTableAxisY1^.Position = #moduleInterface.configuration.Y1Position[16]) AND (#tempAlignTableAxisY2^.Position = #moduleInterface.configuration.Y2Position[16]) THEN
       #moduleInterface.monitoring.alignTableCurrentDeg := -7.0;
   END_IF;
   IF TRUE AND (#tempAlignTableAxisX^.Position = #moduleInterface.configuration.XPosition[17]) AND (#tempAlignTableAxisY1^.Position = #moduleInterface.configuration.Y1Position[17]) AND (#tempAlignTableAxisY2^.Position = #moduleInterface.configuration.Y2Position[17]) THEN
       #moduleInterface.monitoring.alignTableCurrentDeg := -8.0;
   END_IF;
   IF TRUE AND (#tempAlignTableAxisX^.Position = #moduleInterface.configuration.XPosition[18]) AND (#tempAlignTableAxisY1^.Position = #moduleInterface.configuration.Y1Position[18]) AND (#tempAlignTableAxisY2^.Position = #moduleInterface.configuration.Y2Position[18]) THEN
       #moduleInterface.monitoring.alignTableCurrentDeg := -9.0;
   END_IF;
END_REGION
END_FUNCTION_BLOCK
